KUKA KRL program: f1_Kuka_APT217T02S17.SRC

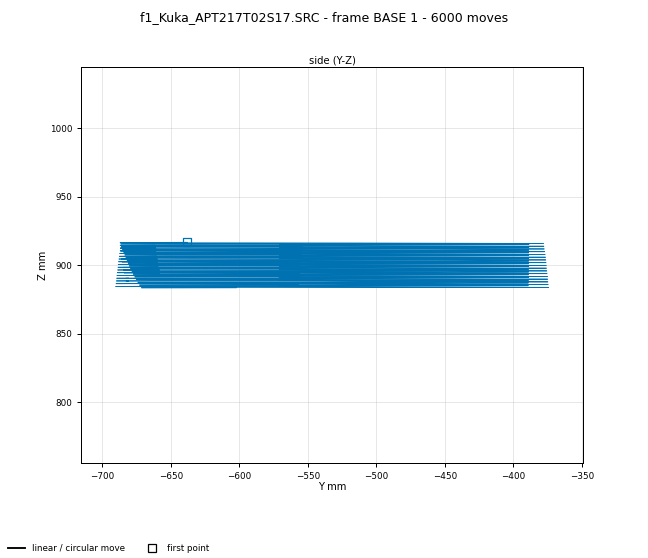
[picture p0: tool path of f1_Kuka_APT217T02S17.SRC in frame BASE 1, 6000 of 6001 moves have a stored position in this frame; points joined in program order, loops and branches not executed]
&ACCESS RVP
&REL 2
&PARAM TEMPLATE = C:\KRC\Roboter\Template\vorgabe
&PARAM EDITMASK = *
DEF f1_Kuka_APT217T02S17()


;FOLD INI;%{PE}%V3.2.0,%MKUKATPBASIS,%CINIT,%VCOMMON,%P
  ;FOLD BAS INI;%{E}%V3.2.0,%MKUKATPBASIS,%CINIT,%VINIT,%P
    GLOBAL INTERRUPT DECL 3 WHEN $STOPMESS==TRUE DO IR_STOPM ( )
    INTERRUPT ON 3
    BAS (#INITMOV,0 )
  ;ENDFOLD (BAS INI)
  ;FOLD USER INI;%{E}%V3.2.0,%MKUKATPUSER,%CINIT,%VINIT,%P
    ;Make your modifications here
  ;ENDFOLD (USER INI)
;ENDFOLD (INI)


;*** Make Null PTP Move
  PTP $pos_act

;*** Auto Load The Correct TOOL Data
  $tool=tool_data[2]

;*** Auto Load The Correct BASE Data
  $base=base_data[1]

  $ADVANCE = 5

;*** Restate Last Velocity
MMPM(30000.0)
SetRPM(8000)
LIN {X -0.126,Y -637.858,Z 916.652,A 0.000,B 0.000,C 90.000,E1 333.384} C_DIS
LIN {X 0.038,Y -640.175,Z 916.648,A 0.000,B 0.000,C 90.000,E1 332.615} C_DIS
LIN {X -0.210,Y -643.727,Z 916.641,A 0.000,B 0.000,C 90.000,E1 331.385} C_DIS
LIN {X 0.321,Y -645.721,Z 916.637,A 0.000,B 0.000,C 90.000,E1 330.589} C_DIS
LIN {X -0.408,Y -648.888,Z 916.630,A 0.000,B 0.000,C 90.000,E1 329.410} C_DIS
LIN {X 0.136,Y -651.837,Z 916.623,A 0.000,B 0.000,C 90.000,E1 328.122} C_DIS
LIN {X 0.289,Y -653.811,Z 916.618,A 0.000,B 0.000,C 90.000,E1 327.120} C_DIS
LIN {X -0.089,Y -655.582,Z 916.612,A 0.000,B 0.000,C 90.000,E1 326.167} C_DIS
LIN {X 0.388,Y -657.387,Z 916.605,A 0.000,B 0.000,C 90.000,E1 324.895} C_DIS
LIN {X 0.431,Y -658.697,Z 916.600,A 0.000,B 0.000,C 90.000,E1 323.909} C_DIS
LIN {X -0.041,Y -659.709,Z 916.594,A 0.000,B 0.000,C 90.000,E1 322.970} C_DIS
LIN {X 0.023,Y -660.733,Z 916.589,A 0.000,B 0.000,C 90.000,E1 321.984} C_DIS
LIN {X -0.032,Y -662.440,Z 916.578,A 0.000,B 0.000,C 90.000,E1 320.033} C_DIS
LIN {X -0.057,Y -664.582,Z 916.564,A 0.000,B 0.000,C 90.000,E1 317.595} C_DIS
LIN {X -0.049,Y -665.667,Z 916.559,A 0.000,B 0.000,C 90.000,E1 316.620} C_DIS
LIN {X -0.059,Y -666.244,Z 916.555,A 0.000,B 0.000,C 90.000,E1 315.891} C_DIS
LIN {X -0.039,Y -668.536,Z 916.540,A 0.000,B 0.000,C 90.000,E1 313.218} C_DIS
LIN {X 0.033,Y -669.951,Z 916.532,A 0.000,B 0.000,C 90.000,E1 311.757} C_DIS
LIN {X 0.126,Y -671.036,Z 916.525,A 0.000,B 0.000,C 90.000,E1 310.539} C_DIS
LIN {X 0.333,Y -672.440,Z 916.516,A 0.000,B 0.000,C 90.000,E1 308.830} C_DIS
LIN {X 0.031,Y -673.306,Z 916.509,A 0.000,B 0.000,C 90.000,E1 307.649} C_DIS
LIN {X 0.276,Y -673.966,Z 916.504,A 0.000,B 0.000,C 90.000,E1 306.664} C_DIS
LIN {X -0.286,Y -674.754,Z 916.495,A 0.000,B 0.000,C 90.000,E1 305.025} C_DIS
LIN {X -0.132,Y -675.681,Z 916.484,A 0.000,B 0.000,C 90.000,E1 303.086} C_DIS
LIN {X -0.151,Y -677.053,Z 916.472,A 0.000,B 0.000,C 90.000,E1 300.924} C_DIS
LIN {X 0.092,Y -679.753,Z 916.456,A 0.000,B 0.000,C 90.000,E1 298.025} C_DIS
LIN {X -0.217,Y -682.675,Z 916.444,A 0.000,B 0.000,C 90.000,E1 295.899} C_DIS
LIN {X -0.081,Y -684.395,Z 916.437,A 0.000,B 0.000,C 90.000,E1 294.695} C_DIS
LIN {X -0.413,Y -685.550,Z 916.432,A 0.000,B 0.000,C 90.000,E1 293.770} C_DIS
LIN {X -0.037,Y -686.075,Z 916.428,A 0.000,B 0.000,C 90.000,E1 293.025} C_DIS
LIN {X 0.393,Y -685.871,Z 916.425,A 0.000,B 0.000,C 90.000,E1 292.514} C_DIS
LIN {X -0.289,Y -685.638,Z 916.424,A 0.000,B 0.000,C 90.000,E1 292.333} C_DIS
LIN {X -0.123,Y -683.879,Z 916.421,A 0.000,B 0.000,C 90.000,E1 291.844} C_DIS
LIN {X 0.084,Y -682.792,Z 916.420,A 0.000,B 0.000,C 90.000,E1 291.589} C_DIS
LIN {X 0.184,Y -681.840,Z 916.419,A 0.000,B 0.000,C 90.000,E1 291.461} C_DIS
LIN {X 0.036,Y -680.423,Z 916.419,A 0.000,B 0.000,C 90.000,E1 291.354} C_DIS
LIN {X -0.276,Y -674.342,Z 916.416,A 0.000,B 0.000,C 90.000,E1 290.972} C_DIS
LIN {X -0.222,Y -664.750,Z 916.414,A 0.000,B 0.000,C 90.000,E1 290.482} C_DIS
LIN {X 0.163,Y -661.931,Z 916.413,A 0.000,B 0.000,C 90.000,E1 290.301} C_DIS
LIN {X 0.103,Y -661.883,Z 916.413,A 0.000,B 0.000,C 90.000,E1 290.301} C_DIS
LIN {X -0.077,Y -661.363,Z 916.412,A 0.000,B 0.000,C 90.000,E1 290.248} C_DIS
LIN {X -0.121,Y -661.335,Z 916.412,A 0.000,B 0.000,C 90.000,E1 290.248} C_DIS
LIN {X -0.189,Y -661.291,Z 916.411,A 0.000,B 0.000,C 90.000,E1 290.066} C_DIS
LIN {X -0.073,Y -661.806,Z 916.410,A 0.000,B 0.000,C 90.000,E1 289.812} C_DIS
LIN {X -0.182,Y -662.452,Z 916.409,A 0.000,B 0.000,C 90.000,E1 289.577} C_DIS
LIN {X -0.112,Y -665.086,Z 916.405,A 0.000,B 0.000,C 90.000,E1 288.960} C_DIS
LIN {X -0.111,Y -669.502,Z 916.401,A 0.000,B 0.000,C 90.000,E1 288.109} C_DIS
LIN {X -0.265,Y -671.949,Z 916.398,A 0.000,B 0.000,C 90.000,E1 287.638} C_DIS
LIN {X -0.202,Y -674.243,Z 916.395,A 0.000,B 0.000,C 90.000,E1 287.149} C_DIS
LIN {X 0.270,Y -677.258,Z 916.391,A 0.000,B 0.000,C 90.000,E1 286.386} C_DIS
LIN {X 0.318,Y -679.580,Z 916.387,A 0.000,B 0.000,C 90.000,E1 285.662} C_DIS
LIN {X 0.202,Y -681.424,Z 916.383,A 0.000,B 0.000,C 90.000,E1 284.954} C_DIS
LIN {X 0.107,Y -682.977,Z 916.379,A 0.000,B 0.000,C 90.000,E1 284.245} C_DIS
LIN {X 0.004,Y -684.701,Z 916.374,A 0.000,B 0.000,C 90.000,E1 283.300} C_DIS
LIN {X -0.084,Y -686.073,Z 916.369,A 0.000,B 0.000,C 90.000,E1 282.355} C_DIS
LIN {X -0.284,Y -686.702,Z 916.365,A 0.000,B 0.000,C 90.000,E1 281.658} C_DIS
LIN {X -0.320,Y -686.990,Z 916.362,A 0.000,B 0.000,C 90.000,E1 281.186} C_DIS
LIN {X 0.316,Y -686.962,Z 916.359,A 0.000,B 0.000,C 90.000,E1 280.658} C_DIS
LIN {X 0.151,Y -686.618,Z 916.357,A 0.000,B 0.000,C 90.000,E1 280.197} C_DIS
LIN {X 0.129,Y -686.308,Z 916.355,A 0.000,B 0.000,C 90.000,E1 279.962} C_DIS
LIN {X -0.035,Y -685.373,Z 916.353,A 0.000,B 0.000,C 90.000,E1 279.500} C_DIS
LIN {X -0.092,Y -683.965,Z 916.350,A 0.000,B 0.000,C 90.000,E1 279.029} C_DIS
LIN {X -0.267,Y -682.163,Z 916.348,A 0.000,B 0.000,C 90.000,E1 278.568} C_DIS
LIN {X 0.174,Y -678.948,Z 916.344,A 0.000,B 0.000,C 90.000,E1 277.814} C_DIS
LIN {X -0.170,Y -674.663,Z 916.339,A 0.000,B 0.000,C 90.000,E1 277.004} C_DIS
LIN {X 0.105,Y -670.562,Z 916.335,A 0.000,B 0.000,C 90.000,E1 276.258} C_DIS
LIN {X -0.152,Y -667.548,Z 916.332,A 0.000,B 0.000,C 90.000,E1 275.796} C_DIS
LIN {X 0.147,Y -663.221,Z 916.329,A 0.000,B 0.000,C 90.000,E1 275.163} C_DIS
LIN {X -0.158,Y -659.457,Z 916.326,A 0.000,B 0.000,C 90.000,E1 274.702} C_DIS
LIN {X 0.118,Y -655.403,Z 916.323,A 0.000,B 0.000,C 90.000,E1 274.188} C_DIS
LIN {X -0.237,Y -650.891,Z 916.321,A 0.000,B 0.000,C 90.000,E1 273.726} C_DIS
LIN {X 0.033,Y -644.710,Z 916.317,A 0.000,B 0.000,C 90.000,E1 273.094} C_DIS
LIN {X 0.003,Y -638.004,Z 916.314,A 0.000,B 0.000,C 90.000,E1 272.522} C_DIS
LIN {X 0.237,Y -630.908,Z 916.311,A 0.000,B 0.000,C 90.000,E1 271.949} C_DIS
LIN {X -0.302,Y -623.315,Z 916.308,A 0.000,B 0.000,C 90.000,E1 271.489} C_DIS
LIN {X -0.112,Y -617.098,Z 916.306,A 0.000,B 0.000,C 90.000,E1 271.088} C_DIS
LIN {X -0.233,Y -610.802,Z 916.304,A 0.000,B 0.000,C 90.000,E1 270.745} C_DIS
LIN {X -0.206,Y -603.986,Z 916.302,A 0.000,B 0.000,C 90.000,E1 270.401} C_DIS
LIN {X 0.120,Y -597.215,Z 916.300,A 0.000,B 0.000,C 90.000,E1 270.057} C_DIS
LIN {X 0.222,Y -591.868,Z 916.299,A 0.000,B 0.000,C 90.000,E1 269.828} C_DIS
LIN {X -0.037,Y -586.277,Z 916.298,A 0.000,B 0.000,C 90.000,E1 269.656} C_DIS
LIN {X 0.001,Y -578.952,Z 916.297,A 0.000,B 0.000,C 90.000,E1 269.427} C_DIS
LIN {X -0.131,Y -571.158,Z 916.296,A 0.000,B 0.000,C 90.000,E1 269.255} C_DIS
LIN {X -0.099,Y -564.308,Z 916.295,A 0.000,B 0.000,C 90.000,E1 269.141} C_DIS
LIN {X -0.044,Y -552.233,Z 916.295,A 0.000,B 0.000,C 90.000,E1 269.026} C_DIS
LIN {X 0.198,Y -548.996,Z 916.294,A 0.000,B 0.000,C 90.000,E1 268.912} C_DIS
LIN {X -0.230,Y -548.179,Z 916.294,A 0.000,B 0.000,C 90.000,E1 268.912} C_DIS
LIN {X -0.086,Y -545.297,Z 916.293,A 0.000,B 0.000,C 90.000,E1 268.682} C_DIS
LIN {X -0.118,Y -545.280,Z 916.293,A 0.000,B 0.000,C 90.000,E1 268.682} C_DIS
LIN {X 0.231,Y -544.006,Z 916.291,A 0.000,B 0.000,C 90.000,E1 268.282} C_DIS
LIN {X -0.084,Y -542.250,Z 916.282,A 0.000,B 0.000,C 90.000,E1 266.788} C_DIS
LIN {X 0.262,Y -540.038,Z 916.266,A 0.000,B 0.000,C 90.000,E1 263.913} C_DIS
LIN {X -0.077,Y -538.982,Z 916.258,A 0.000,B 0.000,C 90.000,E1 262.527} C_DIS
LIN {X 0.094,Y -537.773,Z 916.251,A 0.000,B 0.000,C 90.000,E1 261.084} C_DIS
LIN {X -0.214,Y -536.376,Z 916.243,A 0.000,B 0.000,C 90.000,E1 259.690} C_DIS
LIN {X 0.020,Y -535.047,Z 916.236,A 0.000,B 0.000,C 90.000,E1 258.522} C_DIS
LIN {X -0.191,Y -532.946,Z 916.227,A 0.000,B 0.000,C 90.000,E1 256.825} C_DIS
LIN {X 0.144,Y -531.230,Z 916.219,A 0.000,B 0.000,C 90.000,E1 255.353} C_DIS
LIN {X -0.221,Y -528.389,Z 916.206,A 0.000,B 0.000,C 90.000,E1 253.087} C_DIS
LIN {X 0.146,Y -526.961,Z 916.200,A 0.000,B 0.000,C 90.000,E1 251.891} C_DIS
LIN {X -0.014,Y -524.300,Z 916.188,A 0.000,B 0.000,C 90.000,E1 249.880} C_DIS
LIN {X 0.123,Y -522.391,Z 916.180,A 0.000,B 0.000,C 90.000,E1 248.411} C_DIS
LIN {X 0.264,Y -520.853,Z 916.174,A 0.000,B 0.000,C 90.000,E1 247.230} C_DIS
LIN {X 0.051,Y -518.689,Z 916.166,A 0.000,B 0.000,C 90.000,E1 245.793} C_DIS
LIN {X 0.145,Y -515.996,Z 916.156,A 0.000,B 0.000,C 90.000,E1 244.024} C_DIS
LIN {X -0.062,Y -514.213,Z 916.149,A 0.000,B 0.000,C 90.000,E1 242.871} C_DIS
LIN {X -0.060,Y -511.194,Z 916.139,A 0.000,B 0.000,C 90.000,E1 241.101} C_DIS
LIN {X 0.208,Y -507.461,Z 916.128,A 0.000,B 0.000,C 90.000,E1 238.997} C_DIS
LIN {X 0.052,Y -505.866,Z 916.123,A 0.000,B 0.000,C 90.000,E1 238.122} C_DIS
LIN {X -0.121,Y -504.124,Z 916.118,A 0.000,B 0.000,C 90.000,E1 237.248} C_DIS
LIN {X 0.262,Y -501.504,Z 916.111,A 0.000,B 0.000,C 90.000,E1 236.008} C_DIS
LIN {X 0.068,Y -498.202,Z 916.103,A 0.000,B 0.000,C 90.000,E1 234.529} C_DIS
LIN {X 0.086,Y -492.885,Z 916.090,A 0.000,B 0.000,C 90.000,E1 232.110} C_DIS
LIN {X 0.021,Y -489.445,Z 916.081,A 0.000,B 0.000,C 90.000,E1 230.598} C_DIS
LIN {X -0.038,Y -485.311,Z 916.071,A 0.000,B 0.000,C 90.000,E1 228.771} C_DIS
LIN {X -0.061,Y -480.572,Z 916.059,A 0.000,B 0.000,C 90.000,E1 226.620} C_DIS
LIN {X -0.243,Y -477.858,Z 916.052,A 0.000,B 0.000,C 90.000,E1 225.405} C_DIS
LIN {X -0.014,Y -474.320,Z 916.044,A 0.000,B 0.000,C 90.000,E1 223.824} C_DIS
LIN {X 0.005,Y -469.406,Z 916.031,A 0.000,B 0.000,C 90.000,E1 221.634} C_DIS
LIN {X -0.021,Y -463.936,Z 916.017,A 0.000,B 0.000,C 90.000,E1 219.116} C_DIS
LIN {X 0.037,Y -460.623,Z 916.009,A 0.000,B 0.000,C 90.000,E1 217.523} C_DIS
LIN {X 0.133,Y -456.514,Z 915.998,A 0.000,B 0.000,C 90.000,E1 215.598} C_DIS
LIN {X 0.147,Y -453.128,Z 915.989,A 0.000,B 0.000,C 90.000,E1 213.992} C_DIS
LIN {X -0.157,Y -449.462,Z 915.980,A 0.000,B 0.000,C 90.000,E1 212.418} C_DIS
LIN {X -0.150,Y -445.960,Z 915.971,A 0.000,B 0.000,C 90.000,E1 210.797} C_DIS
LIN {X -0.003,Y -441.643,Z 915.960,A 0.000,B 0.000,C 90.000,E1 208.821} C_DIS
LIN {X -0.035,Y -438.778,Z 915.953,A 0.000,B 0.000,C 90.000,E1 207.513} C_DIS
LIN {X -0.077,Y -434.437,Z 915.942,A 0.000,B 0.000,C 90.000,E1 205.540} C_DIS
LIN {X -0.030,Y -431.536,Z 915.935,A 0.000,B 0.000,C 90.000,E1 204.207} C_DIS
LIN {X 0.166,Y -426.424,Z 915.922,A 0.000,B 0.000,C 90.000,E1 201.844} C_DIS
LIN {X 0.087,Y -422.781,Z 915.912,A 0.000,B 0.000,C 90.000,E1 200.174} C_DIS
LIN {X 0.148,Y -417.354,Z 915.897,A 0.000,B 0.000,C 90.000,E1 197.457} C_DIS
LIN {X -0.115,Y -414.058,Z 915.888,A 0.000,B 0.000,C 90.000,E1 195.788} C_DIS
LIN {X -0.045,Y -410.566,Z 915.878,A 0.000,B 0.000,C 90.000,E1 194.064} C_DIS
LIN {X -0.121,Y -405.687,Z 915.865,A 0.000,B 0.000,C 90.000,E1 191.658} C_DIS
LIN {X -0.011,Y -402.292,Z 915.855,A 0.000,B 0.000,C 90.000,E1 189.905} C_DIS
LIN {X -0.083,Y -397.378,Z 915.841,A 0.000,B 0.000,C 90.000,E1 187.466} C_DIS
LIN {X 0.029,Y -393.315,Z 915.830,A 0.000,B 0.000,C 90.000,E1 185.334} C_DIS
LIN {X -0.085,Y -388.932,Z 915.816,A 0.000,B 0.000,C 90.000,E1 182.865} C_DIS
LIN {X -0.151,Y -385.959,Z 915.806,A 0.000,B 0.000,C 90.000,E1 181.088} C_DIS
LIN {X -0.081,Y -380.437,Z 915.786,A 0.000,B 0.000,C 90.000,E1 177.478} C_DIS
LIN {X -0.056,Y -379.094,Z 915.780,A 0.000,B 0.000,C 90.000,E1 176.388} C_DIS
LIN {X 0.084,Y -378.445,Z 915.776,A 0.000,B 0.000,C 90.000,E1 175.641} C_DIS
LIN {X -0.051,Y -378.213,Z 915.774,A 0.000,B 0.000,C 90.000,E1 175.298} C_DIS
LIN {X 0.044,Y -378.084,Z 915.769,A 0.000,B 0.000,C 90.000,E1 174.375} C_DIS
LIN {X -0.026,Y -378.161,Z 915.768,A 0.000,B 0.000,C 90.000,E1 174.204} C_DIS
LIN {X 0.097,Y -378.414,Z 915.767,A 0.000,B 0.000,C 90.000,E1 173.970} C_DIS
LIN {X -0.077,Y -378.824,Z 915.764,A 0.000,B 0.000,C 90.000,E1 173.451} C_DIS
LIN {X 0.128,Y -379.882,Z 915.761,A 0.000,B 0.000,C 90.000,E1 172.875} C_DIS
LIN {X 0.056,Y -380.113,Z 915.760,A 0.000,B 0.000,C 90.000,E1 172.704} C_DIS
LIN {X -0.023,Y -381.256,Z 915.758,A 0.000,B 0.000,C 90.000,E1 172.356} C_DIS
LIN {X -0.095,Y -381.987,Z 915.757,A 0.000,B 0.000,C 90.000,E1 172.186} C_DIS
LIN {X -0.089,Y -385.404,Z 915.753,A 0.000,B 0.000,C 90.000,E1 171.602} C_DIS
LIN {X -0.159,Y -386.668,Z 915.752,A 0.000,B 0.000,C 90.000,E1 171.432} C_DIS
LIN {X 0.137,Y -391.555,Z 915.749,A 0.000,B 0.000,C 90.000,E1 170.849} C_DIS
LIN {X 0.042,Y -398.395,Z 915.746,A 0.000,B 0.000,C 90.000,E1 170.274} C_DIS
LIN {X 0.183,Y -418.889,Z 915.738,A 0.000,B 0.000,C 90.000,E1 168.870} C_DIS
LIN {X -0.129,Y -426.813,Z 915.735,A 0.000,B 0.000,C 90.000,E1 168.342} C_DIS
LIN {X -0.046,Y -436.131,Z 915.731,A 0.000,B 0.000,C 90.000,E1 167.589} C_DIS
LIN {X 0.118,Y -442.311,Z 915.728,A 0.000,B 0.000,C 90.000,E1 167.061} C_DIS
LIN {X -0.067,Y -455.872,Z 915.722,A 0.000,B 0.000,C 90.000,E1 165.880} C_DIS
LIN {X 0.233,Y -468.313,Z 915.715,A 0.000,B 0.000,C 90.000,E1 164.574} C_DIS
LIN {X -0.018,Y -473.746,Z 915.711,A 0.000,B 0.000,C 90.000,E1 164.031} C_DIS
LIN {X -0.152,Y -484.248,Z 915.705,A 0.000,B 0.000,C 90.000,E1 162.834} C_DIS
LIN {X -0.017,Y -490.256,Z 915.700,A 0.000,B 0.000,C 90.000,E1 162.054} C_DIS
LIN {X -0.074,Y -497.174,Z 915.695,A 0.000,B 0.000,C 90.000,E1 161.148} C_DIS
LIN {X 0.144,Y -502.648,Z 915.691,A 0.000,B 0.000,C 90.000,E1 160.369} C_DIS
LIN {X -0.159,Y -511.136,Z 915.684,A 0.000,B 0.000,C 90.000,E1 159.209} C_DIS
LIN {X -0.112,Y -516.078,Z 915.680,A 0.000,B 0.000,C 90.000,E1 158.465} C_DIS
LIN {X 0.300,Y -522.071,Z 915.675,A 0.000,B 0.000,C 90.000,E1 157.539} C_DIS
LIN {X 0.324,Y -530.498,Z 915.668,A 0.000,B 0.000,C 90.000,E1 156.230} C_DIS
LIN {X -0.124,Y -533.252,Z 915.666,A 0.000,B 0.000,C 90.000,E1 155.845} C_DIS
LIN {X 0.134,Y -537.693,Z 915.662,A 0.000,B 0.000,C 90.000,E1 155.101} C_DIS
LIN {X -0.061,Y -542.155,Z 915.658,A 0.000,B 0.000,C 90.000,E1 154.409} C_DIS
LIN {X -0.101,Y -550.359,Z 915.650,A 0.000,B 0.000,C 90.000,E1 152.999} C_DIS
LIN {X 0.037,Y -552.775,Z 915.648,A 0.000,B 0.000,C 90.000,E1 152.564} C_DIS
LIN {X 0.161,Y -558.858,Z 915.641,A 0.000,B 0.000,C 90.000,E1 151.435} C_DIS
LIN {X 0.009,Y -565.034,Z 915.635,A 0.000,B 0.000,C 90.000,E1 150.205} C_DIS
LIN {X -0.170,Y -570.374,Z 915.628,A 0.000,B 0.000,C 90.000,E1 149.125} C_DIS
LIN {X 0.052,Y -576.717,Z 915.621,A 0.000,B 0.000,C 90.000,E1 147.740} C_DIS
LIN {X 0.187,Y -580.374,Z 915.616,A 0.000,B 0.000,C 90.000,E1 146.914} C_DIS
LIN {X -0.271,Y -585.063,Z 915.610,A 0.000,B 0.000,C 90.000,E1 145.881} C_DIS
LIN {X -0.139,Y -590.655,Z 915.603,A 0.000,B 0.000,C 90.000,E1 144.529} C_DIS
LIN {X 0.359,Y -594.950,Z 915.597,A 0.000,B 0.000,C 90.000,E1 143.417} C_DIS
LIN {X 0.196,Y -600.029,Z 915.590,A 0.000,B 0.000,C 90.000,E1 142.110} C_DIS
LIN {X -0.029,Y -608.431,Z 915.578,A 0.000,B 0.000,C 90.000,E1 140.033} C_DIS
LIN {X -0.159,Y -614.759,Z 915.569,A 0.000,B 0.000,C 90.000,E1 138.485} C_DIS
LIN {X 0.347,Y -620.060,Z 915.562,A 0.000,B 0.000,C 90.000,E1 137.148} C_DIS
LIN {X -0.063,Y -626.543,Z 915.554,A 0.000,B 0.000,C 90.000,E1 135.648} C_DIS
LIN {X 0.206,Y -631.735,Z 915.547,A 0.000,B 0.000,C 90.000,E1 134.352} C_DIS
LIN {X 0.125,Y -636.887,Z 915.540,A 0.000,B 0.000,C 90.000,E1 133.095} C_DIS
LIN {X 0.217,Y -640.998,Z 915.534,A 0.000,B 0.000,C 90.000,E1 132.081} C_DIS
LIN {X -0.142,Y -645.938,Z 915.527,A 0.000,B 0.000,C 90.000,E1 130.862} C_DIS
LIN {X -0.426,Y -650.812,Z 915.520,A 0.000,B 0.000,C 90.000,E1 129.644} C_DIS
LIN {X -0.139,Y -657.437,Z 915.510,A 0.000,B 0.000,C 90.000,E1 127.890} C_DIS
LIN {X -0.143,Y -662.051,Z 915.504,A 0.000,B 0.000,C 90.000,E1 126.664} C_DIS
LIN {X -0.079,Y -666.435,Z 915.497,A 0.000,B 0.000,C 90.000,E1 125.438} C_DIS
LIN {X 0.213,Y -670.660,Z 915.490,A 0.000,B 0.000,C 90.000,E1 124.199} C_DIS
LIN {X 0.057,Y -673.731,Z 915.485,A 0.000,B 0.000,C 90.000,E1 123.245} C_DIS
LIN {X -0.058,Y -676.467,Z 915.479,A 0.000,B 0.000,C 90.000,E1 122.291} C_DIS
LIN {X -0.142,Y -678.905,Z 915.474,A 0.000,B 0.000,C 90.000,E1 121.337} C_DIS
LIN {X -0.205,Y -681.038,Z 915.469,A 0.000,B 0.000,C 90.000,E1 120.384} C_DIS
LIN {X 0.003,Y -682.799,Z 915.463,A 0.000,B 0.000,C 90.000,E1 119.411} C_DIS
LIN {X 0.243,Y -684.380,Z 915.458,A 0.000,B 0.000,C 90.000,E1 118.437} C_DIS
LIN {X 0.287,Y -685.334,Z 915.454,A 0.000,B 0.000,C 90.000,E1 117.719} C_DIS
LIN {X -0.054,Y -686.123,Z 915.449,A 0.000,B 0.000,C 90.000,E1 116.796} C_DIS
LIN {X 0.136,Y -686.609,Z 915.442,A 0.000,B 0.000,C 90.000,E1 115.591} C_DIS
LIN {X 0.113,Y -686.610,Z 915.437,A 0.000,B 0.000,C 90.000,E1 114.643} C_DIS
LIN {X -0.131,Y -686.362,Z 915.433,A 0.000,B 0.000,C 90.000,E1 113.951} C_DIS
LIN {X 0.088,Y -686.187,Z 915.432,A 0.000,B 0.000,C 90.000,E1 113.695} C_DIS
LIN {X 0.251,Y -685.416,Z 915.429,A 0.000,B 0.000,C 90.000,E1 113.206} C_DIS
LIN {X -0.165,Y -684.930,Z 915.428,A 0.000,B 0.000,C 90.000,E1 113.003} C_DIS
LIN {X 0.093,Y -681.933,Z 915.424,A 0.000,B 0.000,C 90.000,E1 112.386} C_DIS
LIN {X -0.064,Y -681.154,Z 915.424,A 0.000,B 0.000,C 90.000,E1 112.280} C_DIS
LIN {X 0.036,Y -679.980,Z 915.423,A 0.000,B 0.000,C 90.000,E1 112.153} C_DIS
LIN {X -0.049,Y -675.165,Z 915.421,A 0.000,B 0.000,C 90.000,E1 111.844} C_DIS
LIN {X 0.343,Y -673.565,Z 915.421,A 0.000,B 0.000,C 90.000,E1 111.716} C_DIS
LIN {X -0.138,Y -671.671,Z 915.420,A 0.000,B 0.000,C 90.000,E1 111.663} C_DIS
LIN {X -0.195,Y -669.497,Z 915.420,A 0.000,B 0.000,C 90.000,E1 111.589} C_DIS
LIN {X 0.075,Y -662.092,Z 915.419,A 0.000,B 0.000,C 90.000,E1 111.408} C_DIS
LIN {X -0.353,Y -659.835,Z 915.419,A 0.000,B 0.000,C 90.000,E1 111.408} C_DIS
LIN {X 0.325,Y -649.462,Z 915.418,A 0.000,B 0.000,C 90.000,E1 111.280} C_DIS
LIN {X -0.137,Y -640.390,Z 915.418,A 0.000,B 0.000,C 90.000,E1 111.280} C_DIS
LIN {X 0.041,Y -633.213,Z 915.418,A 0.000,B 0.000,C 90.000,E1 111.173} C_DIS
LIN {X -0.269,Y -627.334,Z 915.417,A 0.000,B 0.000,C 90.000,E1 111.099} C_DIS
LIN {X 0.265,Y -621.712,Z 915.416,A 0.000,B 0.000,C 90.000,E1 110.918} C_DIS
LIN {X -0.162,Y -614.292,Z 915.415,A 0.000,B 0.000,C 90.000,E1 110.737} C_DIS
LIN {X 0.222,Y -607.266,Z 915.414,A 0.000,B 0.000,C 90.000,E1 110.429} C_DIS
LIN {X 0.126,Y -604.232,Z 915.413,A 0.000,B 0.000,C 90.000,E1 110.301} C_DIS
LIN {X -0.041,Y -597.919,Z 915.411,A 0.000,B 0.000,C 90.000,E1 109.993} C_DIS
LIN {X -0.041,Y -581.000,Z 915.405,A 0.000,B 0.000,C 90.000,E1 108.906} C_DIS
LIN {X 0.321,Y -579.541,Z 915.405,A 0.000,B 0.000,C 90.000,E1 108.779} C_DIS
LIN {X -0.068,Y -572.884,Z 915.403,A 0.000,B 0.000,C 90.000,E1 108.471} C_DIS
LIN {X 0.259,Y -563.917,Z 915.401,A 0.000,B 0.000,C 90.000,E1 108.055} C_DIS
LIN {X 0.007,Y -557.301,Z 915.399,A 0.000,B 0.000,C 90.000,E1 107.819} C_DIS
LIN {X 0.264,Y -555.523,Z 915.398,A 0.000,B 0.000,C 90.000,E1 107.692} C_DIS
LIN {X -0.046,Y -554.039,Z 915.398,A 0.000,B 0.000,C 90.000,E1 107.583} C_DIS
LIN {X -0.085,Y -554.015,Z 915.398,A 0.000,B 0.000,C 90.000,E1 107.583} C_DIS
LIN {X -0.004,Y -553.661,Z 915.396,A 0.000,B 0.000,C 90.000,E1 107.275} C_DIS
LIN {X -0.171,Y -553.838,Z 915.391,A 0.000,B 0.000,C 90.000,E1 106.315} C_DIS
LIN {X -0.087,Y -554.313,Z 915.384,A 0.000,B 0.000,C 90.000,E1 105.190} C_DIS
LIN {X 0.102,Y -555.375,Z 915.372,A 0.000,B 0.000,C 90.000,E1 102.939} C_DIS
LIN {X 0.067,Y -556.899,Z 915.360,A 0.000,B 0.000,C 90.000,E1 100.715} C_DIS
LIN {X 0.238,Y -558.114,Z 915.350,A 0.000,B 0.000,C 90.000,E1 99.029} C_DIS
LIN {X 0.214,Y -559.092,Z 915.343,A 0.000,B 0.000,C 90.000,E1 97.644} C_DIS
LIN {X 0.003,Y -559.681,Z 915.338,A 0.000,B 0.000,C 90.000,E1 96.834} C_DIS
LIN {X 0.170,Y -560.802,Z 915.327,A 0.000,B 0.000,C 90.000,E1 94.878} C_DIS
LIN {X 0.142,Y -561.497,Z 915.320,A 0.000,B 0.000,C 90.000,E1 93.498} C_DIS
LIN {X 0.091,Y -562.172,Z 915.312,A 0.000,B 0.000,C 90.000,E1 92.121} C_DIS
LIN {X 0.151,Y -562.787,Z 915.303,A 0.000,B 0.000,C 90.000,E1 90.458} C_DIS
LIN {X 0.002,Y -563.052,Z 915.297,A 0.000,B 0.000,C 90.000,E1 89.370} C_DIS
LIN {X 0.078,Y -563.406,Z 915.287,A 0.000,B 0.000,C 90.000,E1 87.707} C_DIS
LIN {X -0.045,Y -563.625,Z 915.281,A 0.000,B 0.000,C 90.000,E1 86.617} C_DIS
LIN {X 0.075,Y -563.903,Z 915.272,A 0.000,B 0.000,C 90.000,E1 84.951} C_DIS
LIN {X 0.248,Y -564.169,Z 915.263,A 0.000,B 0.000,C 90.000,E1 83.280} C_DIS
LIN {X -0.062,Y -564.539,Z 915.254,A 0.000,B 0.000,C 90.000,E1 81.659} C_DIS
LIN {X 0.189,Y -565.090,Z 915.245,A 0.000,B 0.000,C 90.000,E1 79.982} C_DIS
LIN {X 0.092,Y -565.820,Z 915.235,A 0.000,B 0.000,C 90.000,E1 78.342} C_DIS
LIN {X 0.189,Y -566.878,Z 915.225,A 0.000,B 0.000,C 90.000,E1 76.408} C_DIS
LIN {X 0.089,Y -567.666,Z 915.217,A 0.000,B 0.000,C 90.000,E1 75.046} C_DIS
LIN {X 0.328,Y -568.516,Z 915.208,A 0.000,B 0.000,C 90.000,E1 73.378} C_DIS
LIN {X 0.033,Y -569.213,Z 915.199,A 0.000,B 0.000,C 90.000,E1 71.764} C_DIS
LIN {X 0.111,Y -569.773,Z 915.190,A 0.000,B 0.000,C 90.000,E1 70.115} C_DIS
LIN {X 0.207,Y -570.193,Z 915.181,A 0.000,B 0.000,C 90.000,E1 68.465} C_DIS
LIN {X -0.007,Y -570.504,Z 915.171,A 0.000,B 0.000,C 90.000,E1 66.847} C_DIS
LIN {X 0.128,Y -570.704,Z 915.161,A 0.000,B 0.000,C 90.000,E1 64.921} C_DIS
LIN {X 0.223,Y -570.771,Z 915.150,A 0.000,B 0.000,C 90.000,E1 62.999} C_DIS
LIN {X 0.151,Y -570.728,Z 915.143,A 0.000,B 0.000,C 90.000,E1 61.641} C_DIS
LIN {X 0.071,Y -570.705,Z 915.135,A 0.000,B 0.000,C 90.000,E1 60.284} C_DIS
LIN {X -0.051,Y -570.523,Z 915.129,A 0.000,B 0.000,C 90.000,E1 59.203} C_DIS
LIN {X -0.289,Y -570.414,Z 915.124,A 0.000,B 0.000,C 90.000,E1 58.408} C_DIS
LIN {X -0.162,Y -569.643,Z 915.115,A 0.000,B 0.000,C 90.000,E1 56.755} C_DIS
LIN {X -0.171,Y -568.940,Z 915.108,A 0.000,B 0.000,C 90.000,E1 55.388} C_DIS
LIN {X -0.123,Y -568.335,Z 915.103,A 0.000,B 0.000,C 90.000,E1 54.562} C_DIS
LIN {X -0.089,Y -567.280,Z 915.097,A 0.000,B 0.000,C 90.000,E1 53.463} C_DIS
LIN {X 0.050,Y -566.019,Z 915.091,A 0.000,B 0.000,C 90.000,E1 52.351} C_DIS
LIN {X 0.059,Y -564.626,Z 915.085,A 0.000,B 0.000,C 90.000,E1 51.251} C_DIS
LIN {X 0.047,Y -562.855,Z 915.079,A 0.000,B 0.000,C 90.000,E1 50.150} C_DIS
LIN {X 0.277,Y -561.369,Z 915.074,A 0.000,B 0.000,C 90.000,E1 49.299} C_DIS
LIN {X 0.037,Y -560.309,Z 915.071,A 0.000,B 0.000,C 90.000,E1 48.771} C_DIS
LIN {X -0.091,Y -557.742,Z 915.065,A 0.000,B 0.000,C 90.000,E1 47.676} C_DIS
LIN {X 0.053,Y -556.318,Z 915.062,A 0.000,B 0.000,C 90.000,E1 47.106} C_DIS
LIN {X -0.191,Y -553.860,Z 915.057,A 0.000,B 0.000,C 90.000,E1 46.296} C_DIS
LIN {X -0.061,Y -551.166,Z 915.052,A 0.000,B 0.000,C 90.000,E1 45.445} C_DIS
LIN {X -0.028,Y -550.233,Z 915.051,A 0.000,B 0.000,C 90.000,E1 45.162} C_DIS
LIN {X -0.327,Y -547.016,Z 915.046,A 0.000,B 0.000,C 90.000,E1 44.352} C_DIS
LIN {X -0.088,Y -544.098,Z 915.042,A 0.000,B 0.000,C 90.000,E1 43.623} C_DIS
LIN {X -0.075,Y -541.595,Z 915.039,A 0.000,B 0.000,C 90.000,E1 43.056} C_DIS
LIN {X -0.263,Y -538.117,Z 915.035,A 0.000,B 0.000,C 90.000,E1 42.366} C_DIS
LIN {X 0.100,Y -535.202,Z 915.032,A 0.000,B 0.000,C 90.000,E1 41.757} C_DIS
LIN {X -0.312,Y -532.038,Z 915.029,A 0.000,B 0.000,C 90.000,E1 41.229} C_DIS
LIN {X 0.164,Y -527.753,Z 915.025,A 0.000,B 0.000,C 90.000,E1 40.458} C_DIS
LIN {X 0.106,Y -524.083,Z 915.022,A 0.000,B 0.000,C 90.000,E1 39.886} C_DIS
LIN {X -0.097,Y -518.344,Z 915.017,A 0.000,B 0.000,C 90.000,E1 39.036} C_DIS
LIN {X -0.090,Y -513.122,Z 915.013,A 0.000,B 0.000,C 90.000,E1 38.302} C_DIS
LIN {X -0.237,Y -508.757,Z 915.010,A 0.000,B 0.000,C 90.000,E1 37.729} C_DIS
LIN {X 0.184,Y -505.350,Z 915.007,A 0.000,B 0.000,C 90.000,E1 37.237} C_DIS
LIN {X -0.025,Y -500.467,Z 915.004,A 0.000,B 0.000,C 90.000,E1 36.664} C_DIS
LIN {X 0.123,Y -496.856,Z 915.001,A 0.000,B 0.000,C 90.000,E1 36.217} C_DIS
LIN {X -0.091,Y -490.347,Z 914.997,A 0.000,B 0.000,C 90.000,E1 35.518} C_DIS
LIN {X -0.203,Y -483.346,Z 914.993,A 0.000,B 0.000,C 90.000,E1 34.818} C_DIS
LIN {X -0.069,Y -477.565,Z 914.990,A 0.000,B 0.000,C 90.000,E1 34.246} C_DIS
LIN {X 0.147,Y -467.323,Z 914.985,A 0.000,B 0.000,C 90.000,E1 33.293} C_DIS
LIN {X 0.192,Y -459.706,Z 914.981,A 0.000,B 0.000,C 90.000,E1 32.625} C_DIS
LIN {X 0.235,Y -447.533,Z 914.976,A 0.000,B 0.000,C 90.000,E1 31.592} C_DIS
LIN {X 0.050,Y -436.600,Z 914.971,A 0.000,B 0.000,C 90.000,E1 30.718} C_DIS
LIN {X 0.059,Y -411.333,Z 914.958,A 0.000,B 0.000,C 90.000,E1 28.487} C_DIS
LIN {X 0.065,Y -403.947,Z 914.954,A 0.000,B 0.000,C 90.000,E1 27.769} C_DIS
LIN {X -0.031,Y -398.103,Z 914.951,A 0.000,B 0.000,C 90.000,E1 27.180} C_DIS
LIN {X 0.052,Y -394.686,Z 914.949,A 0.000,B 0.000,C 90.000,E1 26.744} C_DIS
LIN {X 0.067,Y -391.741,Z 914.946,A 0.000,B 0.000,C 90.000,E1 26.283} C_DIS
LIN {X 0.137,Y -389.672,Z 914.943,A 0.000,B 0.000,C 90.000,E1 25.668} C_DIS
LIN {X -0.100,Y -388.805,Z 914.939,A 0.000,B 0.000,C 90.000,E1 25.079} C_DIS
LIN {X 0.144,Y -388.587,Z 914.935,A 0.000,B 0.000,C 90.000,E1 24.335} C_DIS
LIN {X -0.139,Y -389.455,Z 914.927,A 0.000,B 0.000,C 90.000,E1 22.950} C_DIS
LIN {X -0.173,Y -392.936,Z 914.908,A 0.000,B 0.000,C 90.000,E1 19.396} C_DIS
LIN {X -0.087,Y -396.272,Z 914.892,A 0.000,B 0.000,C 90.000,E1 16.551} C_DIS
LIN {X 0.117,Y -400.358,Z 914.874,A 0.000,B 0.000,C 90.000,E1 13.355} C_DIS
LIN {X -0.183,Y -404.475,Z 914.859,A 0.000,B 0.000,C 90.000,E1 10.602} C_DIS
LIN {X -0.085,Y -409.648,Z 914.841,A 0.000,B 0.000,C 90.000,E1 7.466} C_DIS
LIN {X 0.001,Y -415.369,Z 914.824,A 0.000,B 0.000,C 90.000,E1 4.359} C_DIS
LIN {X 0.172,Y -420.335,Z 914.811,A 0.000,B 0.000,C 90.000,E1 1.949} C_DIS
LIN {X -0.156,Y -426.994,Z 914.795,A 0.000,B 0.000,C 90.000,E1 359.141} C_DIS
LIN {X 0.180,Y -431.388,Z 914.786,A 0.000,B 0.000,C 90.000,E1 357.421} C_DIS
LIN {X -0.138,Y -433.210,Z 914.783,A 0.000,B 0.000,C 90.000,E1 356.963} C_DIS
LIN {X -0.075,Y -433.947,Z 914.782,A 0.000,B 0.000,C 90.000,E1 356.788} C_DIS
LIN {X 0.111,Y -437.101,Z 914.779,A 0.000,B 0.000,C 90.000,E1 356.216} C_DIS
LIN {X -0.203,Y -441.820,Z 914.777,A 0.000,B 0.000,C 90.000,E1 355.812} C_DIS
LIN {X 0.133,Y -442.733,Z 914.776,A 0.000,B 0.000,C 90.000,E1 355.698} C_DIS
LIN {X 0.043,Y -446.815,Z 914.775,A 0.000,B 0.000,C 90.000,E1 355.469} C_DIS
LIN {X 0.014,Y -461.833,Z 914.771,A 0.000,B 0.000,C 90.000,E1 354.780} C_DIS
LIN {X -0.160,Y -478.676,Z 914.766,A 0.000,B 0.000,C 90.000,E1 353.970} C_DIS
LIN {X 0.030,Y -490.195,Z 914.763,A 0.000,B 0.000,C 90.000,E1 353.337} C_DIS
LIN {X 0.108,Y -503.374,Z 914.759,A 0.000,B 0.000,C 90.000,E1 352.591} C_DIS
LIN {X -0.138,Y -509.900,Z 914.757,A 0.000,B 0.000,C 90.000,E1 352.243} C_DIS
LIN {X 0.277,Y -519.398,Z 914.754,A 0.000,B 0.000,C 90.000,E1 351.602} C_DIS
LIN {X -0.205,Y -528.490,Z 914.750,A 0.000,B 0.000,C 90.000,E1 351.027} C_DIS
LIN {X 0.068,Y -535.929,Z 914.747,A 0.000,B 0.000,C 90.000,E1 350.443} C_DIS
LIN {X -0.054,Y -543.007,Z 914.744,A 0.000,B 0.000,C 90.000,E1 349.859} C_DIS
LIN {X 0.086,Y -549.702,Z 914.740,A 0.000,B 0.000,C 90.000,E1 349.218} C_DIS
LIN {X -0.026,Y -554.997,Z 914.737,A 0.000,B 0.000,C 90.000,E1 348.701} C_DIS
LIN {X 0.096,Y -558.836,Z 914.735,A 0.000,B 0.000,C 90.000,E1 348.285} C_DIS
LIN {X 0.187,Y -564.823,Z 914.731,A 0.000,B 0.000,C 90.000,E1 347.589} C_DIS
LIN {X 0.144,Y -571.511,Z 914.727,A 0.000,B 0.000,C 90.000,E1 346.769} C_DIS
LIN {X -0.254,Y -577.653,Z 914.722,A 0.000,B 0.000,C 90.000,E1 345.992} C_DIS
LIN {X -0.170,Y -583.228,Z 914.718,A 0.000,B 0.000,C 90.000,E1 345.172} C_DIS
LIN {X 0.122,Y -588.411,Z 914.713,A 0.000,B 0.000,C 90.000,E1 344.338} C_DIS
LIN {X -0.023,Y -592.424,Z 914.709,A 0.000,B 0.000,C 90.000,E1 343.685} C_DIS
LIN {X -0.263,Y -597.692,Z 914.704,A 0.000,B 0.000,C 90.000,E1 342.779} C_DIS
LIN {X 0.097,Y -605.914,Z 914.695,A 0.000,B 0.000,C 90.000,E1 341.167} C_DIS
LIN {X -0.048,Y -611.653,Z 914.689,A 0.000,B 0.000,C 90.000,E1 340.007} C_DIS
LIN {X -0.109,Y -617.032,Z 914.682,A 0.000,B 0.000,C 90.000,E1 338.847} C_DIS
LIN {X 0.157,Y -620.407,Z 914.678,A 0.000,B 0.000,C 90.000,E1 338.050} C_DIS
LIN {X -0.124,Y -624.708,Z 914.672,A 0.000,B 0.000,C 90.000,E1 337.050} C_DIS
LIN {X -0.346,Y -628.656,Z 914.667,A 0.000,B 0.000,C 90.000,E1 336.049} C_DIS
LIN {X 0.321,Y -632.321,Z 914.661,A 0.000,B 0.000,C 90.000,E1 334.973} C_DIS
LIN {X -0.331,Y -636.659,Z 914.654,A 0.000,B 0.000,C 90.000,E1 333.768} C_DIS
LIN {X -0.180,Y -639.104,Z 914.650,A 0.000,B 0.000,C 90.000,E1 332.999} C_DIS
LIN {X -0.005,Y -641.312,Z 914.646,A 0.000,B 0.000,C 90.000,E1 332.231} C_DIS
LIN {X -0.307,Y -644.146,Z 914.640,A 0.000,B 0.000,C 90.000,E1 331.257} C_DIS
LIN {X -0.181,Y -647.431,Z 914.633,A 0.000,B 0.000,C 90.000,E1 329.999} C_DIS
LIN {X -0.081,Y -649.885,Z 914.628,A 0.000,B 0.000,C 90.000,E1 328.997} C_DIS
LIN {X 0.050,Y -652.253,Z 914.622,A 0.000,B 0.000,C 90.000,E1 327.995} C_DIS
LIN {X 0.116,Y -653.743,Z 914.618,A 0.000,B 0.000,C 90.000,E1 327.248} C_DIS
LIN {X -0.260,Y -655.564,Z 914.613,A 0.000,B 0.000,C 90.000,E1 326.294} C_DIS
LIN {X -0.246,Y -657.070,Z 914.607,A 0.000,B 0.000,C 90.000,E1 325.308} C_DIS
LIN {X -0.207,Y -658.427,Z 914.602,A 0.000,B 0.000,C 90.000,E1 324.322} C_DIS
LIN {X -0.097,Y -659.326,Z 914.598,A 0.000,B 0.000,C 90.000,E1 323.577} C_DIS
LIN {X 0.352,Y -661.057,Z 914.588,A 0.000,B 0.000,C 90.000,E1 321.823} C_DIS
LIN {X -0.088,Y -662.609,Z 914.579,A 0.000,B 0.000,C 90.000,E1 320.150} C_DIS
LIN {X 0.336,Y -664.251,Z 914.568,A 0.000,B 0.000,C 90.000,E1 318.162} C_DIS
LIN {X -0.158,Y -665.848,Z 914.560,A 0.000,B 0.000,C 90.000,E1 316.743} C_DIS
LIN {X 0.318,Y -666.461,Z 914.556,A 0.000,B 0.000,C 90.000,E1 315.972} C_DIS
LIN {X -0.111,Y -668.776,Z 914.541,A 0.000,B 0.000,C 90.000,E1 313.338} C_DIS
LIN {X -0.073,Y -670.177,Z 914.533,A 0.000,B 0.000,C 90.000,E1 311.881} C_DIS
LIN {X 0.016,Y -671.235,Z 914.526,A 0.000,B 0.000,C 90.000,E1 310.663} C_DIS
LIN {X -0.207,Y -672.628,Z 914.517,A 0.000,B 0.000,C 90.000,E1 308.991} C_DIS
LIN {X 0.443,Y -673.517,Z 914.510,A 0.000,B 0.000,C 90.000,E1 307.729} C_DIS
LIN {X 0.153,Y -674.204,Z 914.505,A 0.000,B 0.000,C 90.000,E1 306.790} C_DIS
LIN {X -0.005,Y -674.908,Z 914.496,A 0.000,B 0.000,C 90.000,E1 305.358} C_DIS
LIN {X 0.013,Y -675.599,Z 914.488,A 0.000,B 0.000,C 90.000,E1 303.913} C_DIS
LIN {X -0.005,Y -676.822,Z 914.476,A 0.000,B 0.000,C 90.000,E1 301.750} C_DIS
LIN {X -0.011,Y -679.215,Z 914.460,A 0.000,B 0.000,C 90.000,E1 298.871} C_DIS
LIN {X 0.078,Y -682.521,Z 914.446,A 0.000,B 0.000,C 90.000,E1 296.232} C_DIS
LIN {X -0.188,Y -684.596,Z 914.438,A 0.000,B 0.000,C 90.000,E1 294.823} C_DIS
LIN {X 0.387,Y -685.725,Z 914.433,A 0.000,B 0.000,C 90.000,E1 293.823} C_DIS
LIN {X -0.084,Y -686.143,Z 914.430,A 0.000,B 0.000,C 90.000,E1 293.387} C_DIS
LIN {X 0.079,Y -686.327,Z 914.427,A 0.000,B 0.000,C 90.000,E1 292.898} C_DIS
LIN {X -0.386,Y -686.047,Z 914.425,A 0.000,B 0.000,C 90.000,E1 292.461} C_DIS
LIN {X -0.172,Y -685.510,Z 914.423,A 0.000,B 0.000,C 90.000,E1 292.206} C_DIS
LIN {X -0.217,Y -684.596,Z 914.422,A 0.000,B 0.000,C 90.000,E1 291.972} C_DIS
LIN {X -0.007,Y -683.524,Z 914.421,A 0.000,B 0.000,C 90.000,E1 291.716} C_DIS
LIN {X 0.096,Y -682.876,Z 914.420,A 0.000,B 0.000,C 90.000,E1 291.589} C_DIS
LIN {X 0.197,Y -681.934,Z 914.419,A 0.000,B 0.000,C 90.000,E1 291.461} C_DIS
LIN {X 0.048,Y -680.529,Z 914.419,A 0.000,B 0.000,C 90.000,E1 291.354} C_DIS
LIN {X -0.098,Y -674.324,Z 914.417,A 0.000,B 0.000,C 90.000,E1 290.972} C_DIS
LIN {X -0.074,Y -661.997,Z 914.413,A 0.000,B 0.000,C 90.000,E1 290.355} C_DIS
LIN {X -0.133,Y -661.936,Z 914.413,A 0.000,B 0.000,C 90.000,E1 290.355} C_DIS
LIN {X -0.061,Y -661.178,Z 914.413,A 0.000,B 0.000,C 90.000,E1 290.248} C_DIS
LIN {X -0.104,Y -661.174,Z 914.412,A 0.000,B 0.000,C 90.000,E1 290.248} C_DIS
LIN {X 0.102,Y -661.165,Z 914.411,A 0.000,B 0.000,C 90.000,E1 289.993} C_DIS
LIN {X 0.106,Y -662.558,Z 914.408,A 0.000,B 0.000,C 90.000,E1 289.504} C_DIS
LIN {X 0.016,Y -665.920,Z 914.404,A 0.000,B 0.000,C 90.000,E1 288.779} C_DIS
LIN {X -0.181,Y -670.318,Z 914.400,A 0.000,B 0.000,C 90.000,E1 287.946} C_DIS
LIN {X -0.122,Y -672.691,Z 914.397,A 0.000,B 0.000,C 90.000,E1 287.457} C_DIS
LIN {X -0.254,Y -674.935,Z 914.394,A 0.000,B 0.000,C 90.000,E1 286.985} C_DIS
LIN {X -0.174,Y -676.917,Z 914.392,A 0.000,B 0.000,C 90.000,E1 286.496} C_DIS
LIN {X -0.320,Y -679.336,Z 914.388,A 0.000,B 0.000,C 90.000,E1 285.788} C_DIS
LIN {X -0.259,Y -681.198,Z 914.384,A 0.000,B 0.000,C 90.000,E1 285.064} C_DIS
LIN {X 0.300,Y -682.766,Z 914.380,A 0.000,B 0.000,C 90.000,E1 284.300} C_DIS
LIN {X 0.190,Y -684.519,Z 914.374,A 0.000,B 0.000,C 90.000,E1 283.355} C_DIS
LIN {X 0.121,Y -685.567,Z 914.370,A 0.000,B 0.000,C 90.000,E1 282.647} C_DIS
LIN {X -0.067,Y -686.139,Z 914.368,A 0.000,B 0.000,C 90.000,E1 282.187} C_DIS
LIN {X -0.122,Y -686.734,Z 914.364,A 0.000,B 0.000,C 90.000,E1 281.478} C_DIS
LIN {X -0.142,Y -686.888,Z 914.362,A 0.000,B 0.000,C 90.000,E1 281.243} C_DIS
LIN {X -0.311,Y -686.853,Z 914.360,A 0.000,B 0.000,C 90.000,E1 280.782} C_DIS
LIN {X 0.325,Y -686.567,Z 914.357,A 0.000,B 0.000,C 90.000,E1 280.254} C_DIS
LIN {X 0.303,Y -686.322,Z 914.356,A 0.000,B 0.000,C 90.000,E1 280.018} C_DIS
LIN {X 0.138,Y -685.417,Z 914.353,A 0.000,B 0.000,C 90.000,E1 279.557} C_DIS
LIN {X -0.028,Y -684.045,Z 914.351,A 0.000,B 0.000,C 90.000,E1 279.095} C_DIS
LIN {X -0.096,Y -682.340,Z 914.348,A 0.000,B 0.000,C 90.000,E1 278.624} C_DIS
LIN {X -0.237,Y -681.406,Z 914.347,A 0.000,B 0.000,C 90.000,E1 278.398} C_DIS
LIN {X 0.345,Y -679.252,Z 914.344,A 0.000,B 0.000,C 90.000,E1 277.871} C_DIS
LIN {X -0.005,Y -675.626,Z 914.340,A 0.000,B 0.000,C 90.000,E1 277.182} C_DIS
LIN {X -0.308,Y -672.334,Z 914.337,A 0.000,B 0.000,C 90.000,E1 276.606} C_DIS
LIN {X 0.117,Y -669.462,Z 914.334,A 0.000,B 0.000,C 90.000,E1 276.087} C_DIS
LIN {X -0.060,Y -667.150,Z 914.332,A 0.000,B 0.000,C 90.000,E1 275.739} C_DIS
LIN {X 0.322,Y -663.724,Z 914.329,A 0.000,B 0.000,C 90.000,E1 275.220} C_DIS
LIN {X -0.075,Y -658.987,Z 914.326,A 0.000,B 0.000,C 90.000,E1 274.645} C_DIS
LIN {X 0.230,Y -654.892,Z 914.323,A 0.000,B 0.000,C 90.000,E1 274.131} C_DIS
LIN {X -0.128,Y -650.320,Z 914.320,A 0.000,B 0.000,C 90.000,E1 273.669} C_DIS
LIN {X 0.218,Y -645.416,Z 914.318,A 0.000,B 0.000,C 90.000,E1 273.154} C_DIS
LIN {X 0.160,Y -638.709,Z 914.314,A 0.000,B 0.000,C 90.000,E1 272.579} C_DIS
LIN {X -0.146,Y -631.775,Z 914.311,A 0.000,B 0.000,C 90.000,E1 272.064} C_DIS
LIN {X -0.133,Y -624.238,Z 914.309,A 0.000,B 0.000,C 90.000,E1 271.547} C_DIS
LIN {X -0.014,Y -617.953,Z 914.306,A 0.000,B 0.000,C 90.000,E1 271.146} C_DIS
LIN {X -0.253,Y -611.450,Z 914.304,A 0.000,B 0.000,C 90.000,E1 270.802} C_DIS
LIN {X 0.147,Y -602.987,Z 914.302,A 0.000,B 0.000,C 90.000,E1 270.344} C_DIS
LIN {X 0.091,Y -597.942,Z 914.301,A 0.000,B 0.000,C 90.000,E1 270.115} C_DIS
LIN {X 0.014,Y -590.759,Z 914.299,A 0.000,B 0.000,C 90.000,E1 269.828} C_DIS
LIN {X -0.245,Y -583.097,Z 914.298,A 0.000,B 0.000,C 90.000,E1 269.599} C_DIS
LIN {X -0.125,Y -577.613,Z 914.297,A 0.000,B 0.000,C 90.000,E1 269.427} C_DIS
LIN {X 0.258,Y -571.750,Z 914.296,A 0.000,B 0.000,C 90.000,E1 269.255} C_DIS
LIN {X -0.278,Y -565.008,Z 914.295,A 0.000,B 0.000,C 90.000,E1 269.198} C_DIS
LIN {X -0.084,Y -555.104,Z 914.295,A 0.000,B 0.000,C 90.000,E1 269.083} C_DIS
LIN {X 0.271,Y -552.540,Z 914.295,A 0.000,B 0.000,C 90.000,E1 269.026} C_DIS
LIN {X 0.047,Y -549.313,Z 914.294,A 0.000,B 0.000,C 90.000,E1 268.969} C_DIS
LIN {X -0.042,Y -545.247,Z 914.293,A 0.000,B 0.000,C 90.000,E1 268.682} C_DIS
LIN {X -0.074,Y -545.214,Z 914.293,A 0.000,B 0.000,C 90.000,E1 268.682} C_DIS
LIN {X 0.043,Y -544.194,Z 914.291,A 0.000,B 0.000,C 90.000,E1 268.396} C_DIS
LIN {X -0.134,Y -542.815,Z 914.285,A 0.000,B 0.000,C 90.000,E1 267.364} C_DIS
LIN {X 0.232,Y -540.235,Z 914.268,A 0.000,B 0.000,C 90.000,E1 264.204} C_DIS
LIN {X -0.045,Y -538.992,Z 914.258,A 0.000,B 0.000,C 90.000,E1 262.527} C_DIS
LIN {X 0.126,Y -537.753,Z 914.251,A 0.000,B 0.000,C 90.000,E1 261.084} C_DIS
LIN {X -0.182,Y -536.363,Z 914.243,A 0.000,B 0.000,C 90.000,E1 259.690} C_DIS
LIN {X 0.052,Y -535.069,Z 914.236,A 0.000,B 0.000,C 90.000,E1 258.522} C_DIS
LIN {X -0.160,Y -532.985,Z 914.227,A 0.000,B 0.000,C 90.000,E1 256.825} C_DIS
LIN {X -0.165,Y -530.921,Z 914.217,A 0.000,B 0.000,C 90.000,E1 255.102} C_DIS
LIN {X -0.187,Y -528.419,Z 914.206,A 0.000,B 0.000,C 90.000,E1 253.087} C_DIS
LIN {X 0.180,Y -526.995,Z 914.200,A 0.000,B 0.000,C 90.000,E1 251.891} C_DIS
LIN {X 0.021,Y -524.331,Z 914.188,A 0.000,B 0.000,C 90.000,E1 249.880} C_DIS
LIN {X -0.168,Y -522.058,Z 914.179,A 0.000,B 0.000,C 90.000,E1 248.156} C_DIS
LIN {X -0.027,Y -520.421,Z 914.172,A 0.000,B 0.000,C 90.000,E1 246.975} C_DIS
LIN {X 0.086,Y -518.722,Z 914.166,A 0.000,B 0.000,C 90.000,E1 245.793} C_DIS
LIN {X -0.157,Y -515.633,Z 914.154,A 0.000,B 0.000,C 90.000,E1 243.768} C_DIS
LIN {X 0.088,Y -513.747,Z 914.148,A 0.000,B 0.000,C 90.000,E1 242.564} C_DIS
LIN {X -0.022,Y -511.230,Z 914.139,A 0.000,B 0.000,C 90.000,E1 241.101} C_DIS
LIN {X 0.246,Y -507.503,Z 914.128,A 0.000,B 0.000,C 90.000,E1 238.997} C_DIS
LIN {X 0.091,Y -505.914,Z 914.123,A 0.000,B 0.000,C 90.000,E1 238.122} C_DIS
LIN {X 0.228,Y -503.551,Z 914.116,A 0.000,B 0.000,C 90.000,E1 236.914} C_DIS
LIN {X -0.218,Y -500.309,Z 914.108,A 0.000,B 0.000,C 90.000,E1 235.468} C_DIS
LIN {X -0.180,Y -498.262,Z 914.103,A 0.000,B 0.000,C 90.000,E1 234.562} C_DIS
LIN {X -0.143,Y -494.900,Z 914.095,A 0.000,B 0.000,C 90.000,E1 233.050} C_DIS
LIN {X -0.015,Y -492.290,Z 914.088,A 0.000,B 0.000,C 90.000,E1 231.823} C_DIS
LIN {X 0.217,Y -488.809,Z 914.079,A 0.000,B 0.000,C 90.000,E1 230.275} C_DIS
LIN {X -0.172,Y -484.744,Z 914.069,A 0.000,B 0.000,C 90.000,E1 228.485} C_DIS
LIN {X 0.239,Y -479.320,Z 914.056,A 0.000,B 0.000,C 90.000,E1 225.972} C_DIS
LIN {X 0.150,Y -475.818,Z 914.047,A 0.000,B 0.000,C 90.000,E1 224.433} C_DIS
LIN {X -0.010,Y -472.235,Z 914.038,A 0.000,B 0.000,C 90.000,E1 222.894} C_DIS
LIN {X 0.055,Y -469.437,Z 914.031,A 0.000,B 0.000,C 90.000,E1 221.634} C_DIS
LIN {X 0.030,Y -464.000,Z 914.017,A 0.000,B 0.000,C 90.000,E1 219.116} C_DIS
LIN {X 0.089,Y -460.654,Z 914.009,A 0.000,B 0.000,C 90.000,E1 217.523} C_DIS
LIN {X 0.081,Y -457.245,Z 914.000,A 0.000,B 0.000,C 90.000,E1 215.931} C_DIS
LIN {X 0.199,Y -453.192,Z 913.989,A 0.000,B 0.000,C 90.000,E1 213.992} C_DIS
LIN {X -0.103,Y -449.521,Z 913.980,A 0.000,B 0.000,C 90.000,E1 212.418} C_DIS
LIN {X -0.095,Y -446.025,Z 913.971,A 0.000,B 0.000,C 90.000,E1 210.797} C_DIS
LIN {X 0.052,Y -441.707,Z 913.960,A 0.000,B 0.000,C 90.000,E1 208.821} C_DIS
LIN {X 0.021,Y -438.842,Z 913.953,A 0.000,B 0.000,C 90.000,E1 207.513} C_DIS
LIN {X -0.020,Y -434.500,Z 913.942,A 0.000,B 0.000,C 90.000,E1 205.540} C_DIS
LIN {X 0.028,Y -431.602,Z 913.935,A 0.000,B 0.000,C 90.000,E1 204.207} C_DIS
LIN {X -0.170,Y -426.509,Z 913.922,A 0.000,B 0.000,C 90.000,E1 201.897} C_DIS
LIN {X 0.148,Y -422.872,Z 913.912,A 0.000,B 0.000,C 90.000,E1 200.174} C_DIS
LIN {X 0.048,Y -418.094,Z 913.899,A 0.000,B 0.000,C 90.000,E1 197.819} C_DIS
LIN {X 0.164,Y -415.459,Z 913.892,A 0.000,B 0.000,C 90.000,E1 196.441} C_DIS
LIN {X 0.094,Y -413.438,Z 913.886,A 0.000,B 0.000,C 90.000,E1 195.426} C_DIS
LIN {X 0.046,Y -409.944,Z 913.876,A 0.000,B 0.000,C 90.000,E1 193.716} C_DIS
LIN {X 0.039,Y -405.090,Z 913.863,A 0.000,B 0.000,C 90.000,E1 191.299} C_DIS
LIN {X 0.058,Y -401.673,Z 913.853,A 0.000,B 0.000,C 90.000,E1 189.557} C_DIS
LIN {X -0.011,Y -397.483,Z 913.841,A 0.000,B 0.000,C 90.000,E1 187.466} C_DIS
LIN {X -0.024,Y -392.128,Z 913.826,A 0.000,B 0.000,C 90.000,E1 184.645} C_DIS
LIN {X -0.099,Y -388.412,Z 913.814,A 0.000,B 0.000,C 90.000,E1 182.522} C_DIS
LIN {X -0.073,Y -386.078,Z 913.806,A 0.000,B 0.000,C 90.000,E1 181.088} C_DIS
LIN {X 0.120,Y -381.063,Z 913.788,A 0.000,B 0.000,C 90.000,E1 177.822} C_DIS
LIN {X 0.027,Y -379.120,Z 913.780,A 0.000,B 0.000,C 90.000,E1 176.388} C_DIS
LIN {X 0.168,Y -378.378,Z 913.776,A 0.000,B 0.000,C 90.000,E1 175.641} C_DIS
LIN {X -0.075,Y -377.849,Z 913.772,A 0.000,B 0.000,C 90.000,E1 174.951} C_DIS
LIN {X 0.055,Y -377.701,Z 913.768,A 0.000,B 0.000,C 90.000,E1 174.204} C_DIS
LIN {X -0.197,Y -378.021,Z 913.764,A 0.000,B 0.000,C 90.000,E1 173.514} C_DIS
LIN {X 0.044,Y -378.395,Z 913.763,A 0.000,B 0.000,C 90.000,E1 173.280} C_DIS
LIN {X -0.206,Y -379.451,Z 913.759,A 0.000,B 0.000,C 90.000,E1 172.591} C_DIS
LIN {X 0.114,Y -380.446,Z 913.757,A 0.000,B 0.000,C 90.000,E1 172.186} C_DIS
LIN {X 0.143,Y -381.706,Z 913.755,A 0.000,B 0.000,C 90.000,E1 171.837} C_DIS
LIN {X -0.030,Y -385.985,Z 913.751,A 0.000,B 0.000,C 90.000,E1 171.141} C_DIS
LIN {X 0.115,Y -390.830,Z 913.748,A 0.000,B 0.000,C 90.000,E1 170.566} C_DIS
LIN {X 0.053,Y -397.742,Z 913.744,A 0.000,B 0.000,C 90.000,E1 169.982} C_DIS
LIN {X 0.012,Y -416.133,Z 913.738,A 0.000,B 0.000,C 90.000,E1 168.757} C_DIS
LIN {X 0.210,Y -425.799,Z 913.734,A 0.000,B 0.000,C 90.000,E1 168.049} C_DIS
LIN {X -0.030,Y -435.112,Z 913.730,A 0.000,B 0.000,C 90.000,E1 167.353} C_DIS
LIN {X 0.168,Y -442.765,Z 913.726,A 0.000,B 0.000,C 90.000,E1 166.700} C_DIS
LIN {X -0.105,Y -454.483,Z 913.721,A 0.000,B 0.000,C 90.000,E1 165.700} C_DIS
LIN {X -0.037,Y -461.494,Z 913.717,A 0.000,B 0.000,C 90.000,E1 164.991} C_DIS
LIN {X 0.150,Y -467.129,Z 913.713,A 0.000,B 0.000,C 90.000,E1 164.393} C_DIS
LIN {X -0.001,Y -473.961,Z 913.709,A 0.000,B 0.000,C 90.000,E1 163.685} C_DIS
LIN {X -0.017,Y -481.964,Z 913.704,A 0.000,B 0.000,C 90.000,E1 162.779} C_DIS
LIN {X -0.128,Y -486.972,Z 913.701,A 0.000,B 0.000,C 90.000,E1 162.181} C_DIS
LIN {X 0.113,Y -495.094,Z 913.695,A 0.000,B 0.000,C 90.000,E1 161.094} C_DIS
LIN {X -0.161,Y -500.712,Z 913.691,A 0.000,B 0.000,C 90.000,E1 160.369} C_DIS
LIN {X -0.210,Y -510.342,Z 913.683,A 0.000,B 0.000,C 90.000,E1 159.028} C_DIS
LIN {X 0.008,Y -514.272,Z 913.680,A 0.000,B 0.000,C 90.000,E1 158.411} C_DIS
LIN {X 0.228,Y -521.278,Z 913.674,A 0.000,B 0.000,C 90.000,E1 157.358} C_DIS
LIN {X 0.217,Y -527.029,Z 913.670,A 0.000,B 0.000,C 90.000,E1 156.485} C_DIS
LIN {X -0.217,Y -532.533,Z 913.665,A 0.000,B 0.000,C 90.000,E1 155.665} C_DIS
LIN {X -0.251,Y -538.843,Z 913.659,A 0.000,B 0.000,C 90.000,E1 154.665} C_DIS
LIN {X -0.070,Y -542.267,Z 913.656,A 0.000,B 0.000,C 90.000,E1 154.076} C_DIS
LIN {X 0.269,Y -551.399,Z 913.647,A 0.000,B 0.000,C 90.000,E1 152.487} C_DIS
LIN {X -0.018,Y -555.122,Z 913.643,A 0.000,B 0.000,C 90.000,E1 151.820} C_DIS
LIN {X 0.166,Y -557.472,Z 913.641,A 0.000,B 0.000,C 90.000,E1 151.385} C_DIS
LIN {X 0.268,Y -563.716,Z 913.634,A 0.000,B 0.000,C 90.000,E1 150.127} C_DIS
LIN {X -0.214,Y -569.087,Z 913.628,A 0.000,B 0.000,C 90.000,E1 149.076} C_DIS
LIN {X -0.250,Y -573.613,Z 913.623,A 0.000,B 0.000,C 90.000,E1 148.122} C_DIS
LIN {X -0.073,Y -579.261,Z 913.616,A 0.000,B 0.000,C 90.000,E1 146.882} C_DIS
LIN {X -0.133,Y -584.546,Z 913.609,A 0.000,B 0.000,C 90.000,E1 145.674} C_DIS
LIN {X -0.007,Y -590.206,Z 913.602,A 0.000,B 0.000,C 90.000,E1 144.322} C_DIS
LIN {X 0.267,Y -593.509,Z 913.597,A 0.000,B 0.000,C 90.000,E1 143.497} C_DIS
LIN {X 0.076,Y -598.659,Z 913.590,A 0.000,B 0.000,C 90.000,E1 142.190} C_DIS
LIN {X 0.273,Y -607.086,Z 913.578,A 0.000,B 0.000,C 90.000,E1 140.070} C_DIS
LIN {X 0.054,Y -613.464,Z 913.570,A 0.000,B 0.000,C 90.000,E1 138.528} C_DIS
LIN {X 0.128,Y -618.857,Z 913.563,A 0.000,B 0.000,C 90.000,E1 137.229} C_DIS
LIN {X -0.308,Y -625.315,Z 913.554,A 0.000,B 0.000,C 90.000,E1 135.729} C_DIS
LIN {X 0.059,Y -629.589,Z 913.548,A 0.000,B 0.000,C 90.000,E1 134.676} C_DIS
LIN {X -0.058,Y -634.773,Z 913.541,A 0.000,B 0.000,C 90.000,E1 133.419} C_DIS
LIN {X -0.088,Y -639.945,Z 913.534,A 0.000,B 0.000,C 90.000,E1 132.162} C_DIS
LIN {X -0.041,Y -644.948,Z 913.527,A 0.000,B 0.000,C 90.000,E1 130.906} C_DIS
LIN {X 0.149,Y -649.819,Z 913.520,A 0.000,B 0.000,C 90.000,E1 129.644} C_DIS
LIN {X -0.040,Y -655.482,Z 913.512,A 0.000,B 0.000,C 90.000,E1 128.177} C_DIS
LIN {X -0.075,Y -660.179,Z 913.505,A 0.000,B 0.000,C 90.000,E1 126.950} C_DIS
LIN {X -0.089,Y -662.837,Z 913.501,A 0.000,B 0.000,C 90.000,E1 126.217} C_DIS
LIN {X 0.141,Y -667.154,Z 913.494,A 0.000,B 0.000,C 90.000,E1 124.978} C_DIS
LIN {X 0.317,Y -670.527,Z 913.489,A 0.000,B 0.000,C 90.000,E1 123.992} C_DIS
LIN {X 0.005,Y -672.834,Z 913.485,A 0.000,B 0.000,C 90.000,E1 123.293} C_DIS
LIN {X 0.277,Y -674.953,Z 913.481,A 0.000,B 0.000,C 90.000,E1 122.546} C_DIS
LIN {X 0.171,Y -677.408,Z 913.476,A 0.000,B 0.000,C 90.000,E1 121.592} C_DIS
LIN {X -0.048,Y -678.603,Z 913.473,A 0.000,B 0.000,C 90.000,E1 121.131} C_DIS
LIN {X -0.119,Y -680.622,Z 913.468,A 0.000,B 0.000,C 90.000,E1 120.178} C_DIS
LIN {X 0.082,Y -682.336,Z 913.462,A 0.000,B 0.000,C 90.000,E1 119.205} C_DIS
LIN {X 0.103,Y -683.541,Z 913.458,A 0.000,B 0.000,C 90.000,E1 118.487} C_DIS
LIN {X 0.135,Y -684.518,Z 913.454,A 0.000,B 0.000,C 90.000,E1 117.769} C_DIS
LIN {X 0.081,Y -685.315,Z 913.449,A 0.000,B 0.000,C 90.000,E1 116.821} C_DIS
LIN {X 0.128,Y -685.642,Z 913.445,A 0.000,B 0.000,C 90.000,E1 116.104} C_DIS
LIN {X -0.126,Y -685.937,Z 913.441,A 0.000,B 0.000,C 90.000,E1 115.412} C_DIS
LIN {X 0.066,Y -685.784,Z 913.435,A 0.000,B 0.000,C 90.000,E1 114.207} C_DIS
LIN {X -0.402,Y -685.507,Z 913.432,A 0.000,B 0.000,C 90.000,E1 113.770} C_DIS
LIN {X 0.029,Y -684.757,Z 913.429,A 0.000,B 0.000,C 90.000,E1 113.259} C_DIS
LIN {X -0.027,Y -684.298,Z 913.428,A 0.000,B 0.000,C 90.000,E1 113.025} C_DIS
LIN {X -0.397,Y -681.494,Z 913.425,A 0.000,B 0.000,C 90.000,E1 112.461} C_DIS
LIN {X -0.294,Y -680.757,Z 913.424,A 0.000,B 0.000,C 90.000,E1 112.333} C_DIS
LIN {X -0.196,Y -679.645,Z 913.423,A 0.000,B 0.000,C 90.000,E1 112.206} C_DIS
LIN {X -0.029,Y -676.391,Z 913.422,A 0.000,B 0.000,C 90.000,E1 111.972} C_DIS
LIN {X 0.213,Y -671.943,Z 913.420,A 0.000,B 0.000,C 90.000,E1 111.663} C_DIS
LIN {X -0.008,Y -669.532,Z 913.420,A 0.000,B 0.000,C 90.000,E1 111.589} C_DIS
LIN {X 0.149,Y -666.254,Z 913.419,A 0.000,B 0.000,C 90.000,E1 111.482} C_DIS
LIN {X -0.145,Y -661.500,Z 913.419,A 0.000,B 0.000,C 90.000,E1 111.408} C_DIS
LIN {X 0.041,Y -658.414,Z 913.419,A 0.000,B 0.000,C 90.000,E1 111.354} C_DIS
LIN {X -0.005,Y -648.305,Z 913.418,A 0.000,B 0.000,C 90.000,E1 111.280} C_DIS
LIN {X 0.146,Y -640.639,Z 913.418,A 0.000,B 0.000,C 90.000,E1 111.227} C_DIS
LIN {X -0.053,Y -633.356,Z 913.418,A 0.000,B 0.000,C 90.000,E1 111.153} C_DIS
LIN {X -0.003,Y -627.588,Z 913.417,A 0.000,B 0.000,C 90.000,E1 111.046} C_DIS
LIN {X 0.068,Y -620.234,Z 913.416,A 0.000,B 0.000,C 90.000,E1 110.865} C_DIS
LIN {X -0.224,Y -612.926,Z 913.415,A 0.000,B 0.000,C 90.000,E1 110.663} C_DIS
LIN {X 0.046,Y -605.866,Z 913.413,A 0.000,B 0.000,C 90.000,E1 110.355} C_DIS
LIN {X -0.240,Y -598.211,Z 913.411,A 0.000,B 0.000,C 90.000,E1 109.993} C_DIS
LIN {X -0.257,Y -580.984,Z 913.405,A 0.000,B 0.000,C 90.000,E1 108.906} C_DIS
LIN {X -0.254,Y -577.738,Z 913.404,A 0.000,B 0.000,C 90.000,E1 108.725} C_DIS
LIN {X 0.306,Y -572.805,Z 913.403,A 0.000,B 0.000,C 90.000,E1 108.417} C_DIS
LIN {X 0.157,Y -565.618,Z 913.401,A 0.000,B 0.000,C 90.000,E1 108.127} C_DIS
LIN {X -0.173,Y -557.056,Z 913.399,A 0.000,B 0.000,C 90.000,E1 107.819} C_DIS
LIN {X -0.209,Y -555.920,Z 913.399,A 0.000,B 0.000,C 90.000,E1 107.764} C_DIS
LIN {X -0.148,Y -554.281,Z 913.398,A 0.000,B 0.000,C 90.000,E1 107.583} C_DIS
LIN {X -0.190,Y -554.266,Z 913.398,A 0.000,B 0.000,C 90.000,E1 107.583} C_DIS
LIN {X -0.068,Y -553.877,Z 913.396,A 0.000,B 0.000,C 90.000,E1 107.275} C_DIS
LIN {X -0.116,Y -554.128,Z 913.389,A 0.000,B 0.000,C 90.000,E1 106.024} C_DIS
LIN {X 0.241,Y -554.706,Z 913.381,A 0.000,B 0.000,C 90.000,E1 104.592} C_DIS
LIN {X 0.179,Y -555.726,Z 913.370,A 0.000,B 0.000,C 90.000,E1 102.647} C_DIS
LIN {X 0.053,Y -557.278,Z 913.358,A 0.000,B 0.000,C 90.000,E1 100.433} C_DIS
LIN {X 0.246,Y -558.478,Z 913.349,A 0.000,B 0.000,C 90.000,E1 98.746} C_DIS
LIN {X -0.175,Y -559.674,Z 913.340,A 0.000,B 0.000,C 90.000,E1 97.125} C_DIS
LIN {X -0.086,Y -560.639,Z 913.330,A 0.000,B 0.000,C 90.000,E1 95.454} C_DIS
LIN {X -0.114,Y -561.386,Z 913.323,A 0.000,B 0.000,C 90.000,E1 94.073} C_DIS
LIN {X -0.137,Y -562.050,Z 913.315,A 0.000,B 0.000,C 90.000,E1 92.694} C_DIS
LIN {X -0.184,Y -562.606,Z 913.307,A 0.000,B 0.000,C 90.000,E1 91.318} C_DIS
LIN {X 0.226,Y -562.968,Z 913.301,A 0.000,B 0.000,C 90.000,E1 90.172} C_DIS
LIN {X 0.079,Y -563.221,Z 913.295,A 0.000,B 0.000,C 90.000,E1 89.083} C_DIS
LIN {X 0.054,Y -563.529,Z 913.287,A 0.000,B 0.000,C 90.000,E1 87.707} C_DIS
LIN {X 0.034,Y -563.765,Z 913.280,A 0.000,B 0.000,C 90.000,E1 86.331} C_DIS
LIN {X 0.151,Y -564.059,Z 913.271,A 0.000,B 0.000,C 90.000,E1 84.666} C_DIS
LIN {X 0.230,Y -564.284,Z 913.263,A 0.000,B 0.000,C 90.000,E1 83.280} C_DIS
LIN {X -0.078,Y -564.667,Z 913.254,A 0.000,B 0.000,C 90.000,E1 81.659} C_DIS
LIN {X 0.175,Y -565.215,Z 913.245,A 0.000,B 0.000,C 90.000,E1 79.982} C_DIS
LIN {X 0.081,Y -565.944,Z 913.235,A 0.000,B 0.000,C 90.000,E1 78.342} C_DIS
LIN {X -0.164,Y -566.666,Z 913.228,A 0.000,B 0.000,C 90.000,E1 76.992} C_DIS
LIN {X -0.089,Y -567.617,Z 913.219,A 0.000,B 0.000,C 90.000,E1 75.338} C_DIS
LIN {X -0.005,Y -568.443,Z 913.209,A 0.000,B 0.000,C 90.000,E1 73.685} C_DIS
LIN {X -0.133,Y -569.180,Z 913.200,A 0.000,B 0.000,C 90.000,E1 72.054} C_DIS
LIN {X -0.046,Y -569.646,Z 913.193,A 0.000,B 0.000,C 90.000,E1 70.678} C_DIS
LIN {X -0.108,Y -570.026,Z 913.185,A 0.000,B 0.000,C 90.000,E1 69.316} C_DIS
LIN {X 0.168,Y -570.343,Z 913.177,A 0.000,B 0.000,C 90.000,E1 67.922} C_DIS
LIN {X 0.118,Y -570.557,Z 913.170,A 0.000,B 0.000,C 90.000,E1 66.561} C_DIS
LIN {X -0.042,Y -570.734,Z 913.159,A 0.000,B 0.000,C 90.000,E1 64.665} C_DIS
LIN {X 0.224,Y -570.756,Z 913.150,A 0.000,B 0.000,C 90.000,E1 62.999} C_DIS
LIN {X 0.321,Y -570.774,Z 913.144,A 0.000,B 0.000,C 90.000,E1 61.897} C_DIS
LIN {X 0.071,Y -570.659,Z 913.135,A 0.000,B 0.000,C 90.000,E1 60.284} C_DIS
LIN {X 0.123,Y -570.543,Z 913.130,A 0.000,B 0.000,C 90.000,E1 59.459} C_DIS
LIN {X -0.290,Y -570.328,Z 913.124,A 0.000,B 0.000,C 90.000,E1 58.408} C_DIS
LIN {X -0.289,Y -569.678,Z 913.117,A 0.000,B 0.000,C 90.000,E1 57.041} C_DIS
LIN {X -0.105,Y -569.109,Z 913.111,A 0.000,B 0.000,C 90.000,E1 55.928} C_DIS
LIN {X -0.050,Y -568.598,Z 913.106,A 0.000,B 0.000,C 90.000,E1 55.102} C_DIS
LIN {X -0.129,Y -568.204,Z 913.103,A 0.000,B 0.000,C 90.000,E1 54.562} C_DIS
LIN {X -0.097,Y -567.135,Z 913.097,A 0.000,B 0.000,C 90.000,E1 53.463} C_DIS
LIN {X 0.039,Y -565.855,Z 913.091,A 0.000,B 0.000,C 90.000,E1 52.351} C_DIS
LIN {X 0.047,Y -564.431,Z 913.085,A 0.000,B 0.000,C 90.000,E1 51.251} C_DIS
LIN {X -0.070,Y -563.141,Z 913.080,A 0.000,B 0.000,C 90.000,E1 50.436} C_DIS
LIN {X 0.259,Y -561.119,Z 913.074,A 0.000,B 0.000,C 90.000,E1 49.299} C_DIS
LIN {X 0.018,Y -560.044,Z 913.071,A 0.000,B 0.000,C 90.000,E1 48.771} C_DIS
LIN {X 0.223,Y -558.130,Z 913.066,A 0.000,B 0.000,C 90.000,E1 47.919} C_DIS
LIN {X -0.040,Y -556.769,Z 913.063,A 0.000,B 0.000,C 90.000,E1 47.391} C_DIS
LIN {X 0.126,Y -554.364,Z 913.059,A 0.000,B 0.000,C 90.000,E1 46.539} C_DIS
LIN {X -0.134,Y -551.686,Z 913.054,A 0.000,B 0.000,C 90.000,E1 45.729} C_DIS
LIN {X -0.060,Y -549.792,Z 913.051,A 0.000,B 0.000,C 90.000,E1 45.162} C_DIS
LIN {X 0.018,Y -546.535,Z 913.046,A 0.000,B 0.000,C 90.000,E1 44.312} C_DIS
LIN {X 0.067,Y -542.935,Z 913.042,A 0.000,B 0.000,C 90.000,E1 43.461} C_DIS
LIN {X 0.068,Y -540.325,Z 913.038,A 0.000,B 0.000,C 90.000,E1 42.894} C_DIS
LIN {X 0.083,Y -537.529,Z 913.035,A 0.000,B 0.000,C 90.000,E1 42.324} C_DIS
LIN {X 0.043,Y -534.530,Z 913.032,A 0.000,B 0.000,C 90.000,E1 41.757} C_DIS
LIN {X -0.022,Y -531.304,Z 913.029,A 0.000,B 0.000,C 90.000,E1 41.191} C_DIS
LIN {X 0.097,Y -526.966,Z 913.025,A 0.000,B 0.000,C 90.000,E1 40.458} C_DIS
LIN {X 0.220,Y -524.230,Z 913.022,A 0.000,B 0.000,C 90.000,E1 40.011} C_DIS
LIN {X -0.177,Y -517.457,Z 913.017,A 0.000,B 0.000,C 90.000,E1 39.036} C_DIS
LIN {X -0.057,Y -511.072,Z 913.012,A 0.000,B 0.000,C 90.000,E1 38.141} C_DIS
LIN {X 0.002,Y -505.495,Z 913.008,A 0.000,B 0.000,C 90.000,E1 37.397} C_DIS
LIN {X -0.109,Y -499.310,Z 913.004,A 0.000,B 0.000,C 90.000,E1 36.664} C_DIS
LIN {X -0.141,Y -495.424,Z 913.001,A 0.000,B 0.000,C 90.000,E1 36.217} C_DIS
LIN {X -0.095,Y -490.245,Z 912.998,A 0.000,B 0.000,C 90.000,E1 35.644} C_DIS
LIN {X 0.185,Y -483.249,Z 912.994,A 0.000,B 0.000,C 90.000,E1 34.898} C_DIS
LIN {X 0.037,Y -477.453,Z 912.991,A 0.000,B 0.000,C 90.000,E1 34.358} C_DIS
LIN {X 0.074,Y -467.069,Z 912.986,A 0.000,B 0.000,C 90.000,E1 33.420} C_DIS
LIN {X 0.153,Y -459.489,Z 912.982,A 0.000,B 0.000,C 90.000,E1 32.752} C_DIS
LIN {X -0.084,Y -447.212,Z 912.976,A 0.000,B 0.000,C 90.000,E1 31.750} C_DIS
LIN {X -0.009,Y -436.314,Z 912.971,A 0.000,B 0.000,C 90.000,E1 30.846} C_DIS
LIN {X 0.153,Y -419.894,Z 912.964,A 0.000,B 0.000,C 90.000,E1 29.411} C_DIS
LIN {X 0.200,Y -405.235,Z 912.956,A 0.000,B 0.000,C 90.000,E1 28.025} C_DIS
LIN {X -0.065,Y -397.929,Z 912.952,A 0.000,B 0.000,C 90.000,E1 27.308} C_DIS
LIN {X 0.197,Y -394.754,Z 912.950,A 0.000,B 0.000,C 90.000,E1 26.873} C_DIS
LIN {X -0.017,Y -391.580,Z 912.947,A 0.000,B 0.000,C 90.000,E1 26.411} C_DIS
LIN {X 0.197,Y -389.784,Z 912.944,A 0.000,B 0.000,C 90.000,E1 25.848} C_DIS
LIN {X -0.031,Y -388.753,Z 912.939,A 0.000,B 0.000,C 90.000,E1 25.079} C_DIS
LIN {X 0.026,Y -388.630,Z 912.937,A 0.000,B 0.000,C 90.000,E1 24.719} C_DIS
LIN {X 0.062,Y -389.038,Z 912.931,A 0.000,B 0.000,C 90.000,E1 23.643} C_DIS
LIN {X -0.166,Y -392.681,Z 912.910,A 0.000,B 0.000,C 90.000,E1 19.758} C_DIS
LIN {X -0.088,Y -395.951,Z 912.894,A 0.000,B 0.000,C 90.000,E1 16.913} C_DIS
LIN {X 0.093,Y -398.571,Z 912.882,A 0.000,B 0.000,C 90.000,E1 14.773} C_DIS
LIN {X -0.152,Y -401.482,Z 912.870,A 0.000,B 0.000,C 90.000,E1 12.703} C_DIS
LIN {X -0.108,Y -405.129,Z 912.857,A 0.000,B 0.000,C 90.000,E1 10.254} C_DIS
LIN {X -0.008,Y -409.748,Z 912.841,A 0.000,B 0.000,C 90.000,E1 7.466} C_DIS
LIN {X 0.081,Y -414.776,Z 912.826,A 0.000,B 0.000,C 90.000,E1 4.702} C_DIS
LIN {X -0.163,Y -420.433,Z 912.811,A 0.000,B 0.000,C 90.000,E1 2.007} C_DIS
LIN {X -0.036,Y -428.799,Z 912.791,A 0.000,B 0.000,C 90.000,E1 358.453} C_DIS
LIN {X 0.184,Y -431.460,Z 912.786,A 0.000,B 0.000,C 90.000,E1 357.421} C_DIS
LIN {X -0.073,Y -433.883,Z 912.782,A 0.000,B 0.000,C 90.000,E1 356.788} C_DIS
LIN {X -0.077,Y -436.280,Z 912.780,A 0.000,B 0.000,C 90.000,E1 356.331} C_DIS
LIN {X 0.038,Y -437.286,Z 912.779,A 0.000,B 0.000,C 90.000,E1 356.159} C_DIS
LIN {X 0.077,Y -442.593,Z 912.776,A 0.000,B 0.000,C 90.000,E1 355.641} C_DIS
LIN {X 0.100,Y -448.497,Z 912.774,A 0.000,B 0.000,C 90.000,E1 355.298} C_DIS
LIN {X -0.119,Y -461.754,Z 912.771,A 0.000,B 0.000,C 90.000,E1 354.723} C_DIS
LIN {X 0.100,Y -475.255,Z 912.767,A 0.000,B 0.000,C 90.000,E1 354.033} C_DIS
LIN {X 0.196,Y -488.488,Z 912.763,A 0.000,B 0.000,C 90.000,E1 353.337} C_DIS
LIN {X -0.151,Y -501.551,Z 912.759,A 0.000,B 0.000,C 90.000,E1 352.648} C_DIS
LIN {X 0.172,Y -508.032,Z 912.757,A 0.000,B 0.000,C 90.000,E1 352.243} C_DIS
LIN {X 0.102,Y -517.582,Z 912.754,A 0.000,B 0.000,C 90.000,E1 351.659} C_DIS
LIN {X 0.195,Y -526.813,Z 912.750,A 0.000,B 0.000,C 90.000,E1 351.027} C_DIS
LIN {X -0.020,Y -534.327,Z 912.747,A 0.000,B 0.000,C 90.000,E1 350.500} C_DIS
LIN {X -0.156,Y -541.465,Z 912.744,A 0.000,B 0.000,C 90.000,E1 349.926} C_DIS
LIN {X 0.025,Y -548.243,Z 912.741,A 0.000,B 0.000,C 90.000,E1 349.285} C_DIS
LIN {X 0.050,Y -554.777,Z 912.737,A 0.000,B 0.000,C 90.000,E1 348.634} C_DIS
LIN {X 0.082,Y -558.670,Z 912.735,A 0.000,B 0.000,C 90.000,E1 348.229} C_DIS
LIN {X 0.294,Y -564.641,Z 912.731,A 0.000,B 0.000,C 90.000,E1 347.521} C_DIS
LIN {X 0.006,Y -572.461,Z 912.726,A 0.000,B 0.000,C 90.000,E1 346.589} C_DIS
LIN {X -0.276,Y -577.539,Z 912.722,A 0.000,B 0.000,C 90.000,E1 345.936} C_DIS
LIN {X 0.050,Y -582.216,Z 912.718,A 0.000,B 0.000,C 90.000,E1 345.227} C_DIS
LIN {X -0.146,Y -586.648,Z 912.714,A 0.000,B 0.000,C 90.000,E1 344.574} C_DIS
LIN {X 0.186,Y -591.629,Z 912.710,A 0.000,B 0.000,C 90.000,E1 343.740} C_DIS
LIN {X -0.297,Y -597.672,Z 912.704,A 0.000,B 0.000,C 90.000,E1 342.725} C_DIS
LIN {X 0.004,Y -603.868,Z 912.697,A 0.000,B 0.000,C 90.000,E1 341.511} C_DIS
LIN {X -0.022,Y -607.233,Z 912.694,A 0.000,B 0.000,C 90.000,E1 340.859} C_DIS
LIN {X -0.120,Y -612.312,Z 912.688,A 0.000,B 0.000,C 90.000,E1 339.826} C_DIS
LIN {X 0.067,Y -617.105,Z 912.682,A 0.000,B 0.000,C 90.000,E1 338.773} C_DIS
LIN {X 0.338,Y -620.503,Z 912.678,A 0.000,B 0.000,C 90.000,E1 337.975} C_DIS
LIN {X 0.069,Y -623.798,Z 912.674,A 0.000,B 0.000,C 90.000,E1 337.230} C_DIS
LIN {X -0.161,Y -627.823,Z 912.668,A 0.000,B 0.000,C 90.000,E1 336.230} C_DIS
LIN {X -0.340,Y -631.563,Z 912.662,A 0.000,B 0.000,C 90.000,E1 335.229} C_DIS
LIN {X -0.159,Y -635.997,Z 912.655,A 0.000,B 0.000,C 90.000,E1 333.948} C_DIS
LIN {X 0.046,Y -639.273,Z 912.650,A 0.000,B 0.000,C 90.000,E1 332.922} C_DIS
LIN {X 0.291,Y -642.226,Z 912.644,A 0.000,B 0.000,C 90.000,E1 331.897} C_DIS
LIN {X 0.005,Y -645.038,Z 912.638,A 0.000,B 0.000,C 90.000,E1 330.923} C_DIS
LIN {X 0.150,Y -648.289,Z 912.632,A 0.000,B 0.000,C 90.000,E1 329.665} C_DIS
LIN {X 0.262,Y -650.700,Z 912.626,A 0.000,B 0.000,C 90.000,E1 328.663} C_DIS
LIN {X -0.147,Y -653.029,Z 912.621,A 0.000,B 0.000,C 90.000,E1 327.709} C_DIS
LIN {X -0.436,Y -655.364,Z 912.614,A 0.000,B 0.000,C 90.000,E1 326.501} C_DIS
LIN {X 0.115,Y -656.981,Z 912.608,A 0.000,B 0.000,C 90.000,E1 325.468} C_DIS
LIN {X -0.300,Y -658.684,Z 912.601,A 0.000,B 0.000,C 90.000,E1 324.276} C_DIS
LIN {X 0.147,Y -659.850,Z 912.596,A 0.000,B 0.000,C 90.000,E1 323.256} C_DIS
LIN {X -0.270,Y -661.337,Z 912.588,A 0.000,B 0.000,C 90.000,E1 321.823} C_DIS
LIN {X 0.229,Y -662.935,Z 912.578,A 0.000,B 0.000,C 90.000,E1 320.070} C_DIS
LIN {X 0.200,Y -665.111,Z 912.565,A 0.000,B 0.000,C 90.000,E1 317.634} C_DIS
LIN {X -0.277,Y -666.137,Z 912.559,A 0.000,B 0.000,C 90.000,E1 316.701} C_DIS
LIN {X -0.283,Y -666.754,Z 912.555,A 0.000,B 0.000,C 90.000,E1 315.972} C_DIS
LIN {X -0.259,Y -668.421,Z 912.544,A 0.000,B 0.000,C 90.000,E1 314.028} C_DIS
LIN {X 0.260,Y -669.589,Z 912.538,A 0.000,B 0.000,C 90.000,E1 312.771} C_DIS
LIN {X -0.150,Y -670.716,Z 912.531,A 0.000,B 0.000,C 90.000,E1 311.595} C_DIS
LIN {X -0.054,Y -671.581,Z 912.526,A 0.000,B 0.000,C 90.000,E1 310.620} C_DIS
LIN {X 0.167,Y -672.973,Z 912.516,A 0.000,B 0.000,C 90.000,E1 308.910} C_DIS
LIN {X 0.409,Y -674.061,Z 912.508,A 0.000,B 0.000,C 90.000,E1 307.443} C_DIS
LIN {X 0.125,Y -674.673,Z 912.503,A 0.000,B 0.000,C 90.000,E1 306.503} C_DIS
LIN {X 0.124,Y -675.490,Z 912.494,A 0.000,B 0.000,C 90.000,E1 304.818} C_DIS
LIN {X -0.003,Y -676.069,Z 912.487,A 0.000,B 0.000,C 90.000,E1 303.627} C_DIS
LIN {X -0.191,Y -677.184,Z 912.476,A 0.000,B 0.000,C 90.000,E1 301.720} C_DIS
LIN {X 0.258,Y -679.140,Z 912.463,A 0.000,B 0.000,C 90.000,E1 299.283} C_DIS
LIN {X -0.037,Y -682.604,Z 912.447,A 0.000,B 0.000,C 90.000,E1 296.437} C_DIS
LIN {X -0.077,Y -685.001,Z 912.438,A 0.000,B 0.000,C 90.000,E1 294.771} C_DIS
LIN {X -0.119,Y -686.084,Z 912.432,A 0.000,B 0.000,C 90.000,E1 293.823} C_DIS
LIN {X 0.041,Y -686.462,Z 912.430,A 0.000,B 0.000,C 90.000,E1 293.334} C_DIS
LIN {X -0.423,Y -686.599,Z 912.427,A 0.000,B 0.000,C 90.000,E1 292.898} C_DIS
LIN {X 0.009,Y -686.253,Z 912.424,A 0.000,B 0.000,C 90.000,E1 292.386} C_DIS
LIN {X -0.036,Y -685.610,Z 912.423,A 0.000,B 0.000,C 90.000,E1 292.153} C_DIS
LIN {X 0.176,Y -684.585,Z 912.422,A 0.000,B 0.000,C 90.000,E1 291.897} C_DIS
LIN {X 0.132,Y -683.381,Z 912.420,A 0.000,B 0.000,C 90.000,E1 291.663} C_DIS
LIN {X 0.235,Y -682.660,Z 912.420,A 0.000,B 0.000,C 90.000,E1 291.535} C_DIS
LIN {X 0.336,Y -681.587,Z 912.419,A 0.000,B 0.000,C 90.000,E1 291.408} C_DIS
LIN {X -0.199,Y -679.979,Z 912.418,A 0.000,B 0.000,C 90.000,E1 291.334} C_DIS
LIN {X 0.151,Y -676.328,Z 912.417,A 0.000,B 0.000,C 90.000,E1 291.099} C_DIS
LIN {X 0.153,Y -673.473,Z 912.416,A 0.000,B 0.000,C 90.000,E1 290.918} C_DIS
LIN {X -0.184,Y -665.144,Z 912.414,A 0.000,B 0.000,C 90.000,E1 290.556} C_DIS
LIN {X 0.062,Y -661.702,Z 912.413,A 0.000,B 0.000,C 90.000,E1 290.355} C_DIS
LIN {X 0.003,Y -661.633,Z 912.413,A 0.000,B 0.000,C 90.000,E1 290.355} C_DIS
LIN {X 0.237,Y -660.979,Z 912.413,A 0.000,B 0.000,C 90.000,E1 290.248} C_DIS
LIN {X 0.177,Y -660.944,Z 912.413,A 0.000,B 0.000,C 90.000,E1 290.248} C_DIS
LIN {X -0.061,Y -660.915,Z 912.412,A 0.000,B 0.000,C 90.000,E1 290.120} C_DIS
LIN {X -0.004,Y -661.039,Z 912.411,A 0.000,B 0.000,C 90.000,E1 289.993} C_DIS
LIN {X -0.162,Y -662.096,Z 912.409,A 0.000,B 0.000,C 90.000,E1 289.631} C_DIS
LIN {X -0.119,Y -665.219,Z 912.405,A 0.000,B 0.000,C 90.000,E1 288.906} C_DIS
LIN {X -0.258,Y -670.268,Z 912.400,A 0.000,B 0.000,C 90.000,E1 287.946} C_DIS
LIN {X -0.201,Y -672.645,Z 912.397,A 0.000,B 0.000,C 90.000,E1 287.457} C_DIS
LIN {X -0.136,Y -674.881,Z 912.394,A 0.000,B 0.000,C 90.000,E1 286.968} C_DIS
LIN {X -0.254,Y -676.865,Z 912.392,A 0.000,B 0.000,C 90.000,E1 286.496} C_DIS
LIN {X -0.400,Y -679.268,Z 912.388,A 0.000,B 0.000,C 90.000,E1 285.788} C_DIS
LIN {X 0.316,Y -681.121,Z 912.384,A 0.000,B 0.000,C 90.000,E1 285.009} C_DIS
LIN {X 0.217,Y -682.663,Z 912.380,A 0.000,B 0.000,C 90.000,E1 284.300} C_DIS
LIN {X 0.132,Y -684.038,Z 912.376,A 0.000,B 0.000,C 90.000,E1 283.592} C_DIS
LIN {X 0.059,Y -685.144,Z 912.372,A 0.000,B 0.000,C 90.000,E1 282.883} C_DIS
LIN {X -0.007,Y -686.026,Z 912.368,A 0.000,B 0.000,C 90.000,E1 282.175} C_DIS
LIN {X -0.209,Y -686.613,Z 912.364,A 0.000,B 0.000,C 90.000,E1 281.478} C_DIS
LIN {X -0.229,Y -686.735,Z 912.362,A 0.000,B 0.000,C 90.000,E1 281.243} C_DIS
LIN {X 0.277,Y -686.699,Z 912.360,A 0.000,B 0.000,C 90.000,E1 280.725} C_DIS
LIN {X 0.236,Y -686.392,Z 912.357,A 0.000,B 0.000,C 90.000,E1 280.254} C_DIS
LIN {X 0.214,Y -686.117,Z 912.356,A 0.000,B 0.000,C 90.000,E1 280.018} C_DIS
LIN {X 0.047,Y -685.213,Z 912.353,A 0.000,B 0.000,C 90.000,E1 279.557} C_DIS
LIN {X -0.120,Y -683.886,Z 912.351,A 0.000,B 0.000,C 90.000,E1 279.095} C_DIS
LIN {X -0.189,Y -682.197,Z 912.348,A 0.000,B 0.000,C 90.000,E1 278.624} C_DIS
LIN {X -0.329,Y -681.272,Z 912.347,A 0.000,B 0.000,C 90.000,E1 278.398} C_DIS
LIN {X 0.252,Y -679.114,Z 912.344,A 0.000,B 0.000,C 90.000,E1 277.871} C_DIS
LIN {X -0.026,Y -676.151,Z 912.341,A 0.000,B 0.000,C 90.000,E1 277.296} C_DIS
LIN {X -0.323,Y -672.911,Z 912.337,A 0.000,B 0.000,C 90.000,E1 276.720} C_DIS
LIN {X 0.104,Y -670.092,Z 912.335,A 0.000,B 0.000,C 90.000,E1 276.201} C_DIS
LIN {X -0.072,Y -667.866,Z 912.333,A 0.000,B 0.000,C 90.000,E1 275.853} C_DIS
LIN {X 0.227,Y -663.595,Z 912.329,A 0.000,B 0.000,C 90.000,E1 275.220} C_DIS
LIN {X -0.076,Y -659.873,Z 912.326,A 0.000,B 0.000,C 90.000,E1 274.759} C_DIS
LIN {X 0.103,Y -654.690,Z 912.323,A 0.000,B 0.000,C 90.000,E1 274.131} C_DIS
LIN {X -0.256,Y -650.065,Z 912.320,A 0.000,B 0.000,C 90.000,E1 273.669} C_DIS
LIN {X 0.087,Y -645.130,Z 912.318,A 0.000,B 0.000,C 90.000,E1 273.154} C_DIS
LIN {X 0.054,Y -638.415,Z 912.314,A 0.000,B 0.000,C 90.000,E1 272.579} C_DIS
LIN {X 0.305,Y -631.334,Z 912.311,A 0.000,B 0.000,C 90.000,E1 272.007} C_DIS
LIN {X -0.258,Y -623.770,Z 912.309,A 0.000,B 0.000,C 90.000,E1 271.547} C_DIS
LIN {X -0.102,Y -617.527,Z 912.306,A 0.000,B 0.000,C 90.000,E1 271.146} C_DIS
LIN {X -0.134,Y -611.229,Z 912.304,A 0.000,B 0.000,C 90.000,E1 270.802} C_DIS
LIN {X 0.266,Y -602.692,Z 912.302,A 0.000,B 0.000,C 90.000,E1 270.344} C_DIS
LIN {X 0.213,Y -597.636,Z 912.301,A 0.000,B 0.000,C 90.000,E1 270.115} C_DIS
LIN {X 0.149,Y -590.260,Z 912.299,A 0.000,B 0.000,C 90.000,E1 269.828} C_DIS
LIN {X -0.010,Y -584.798,Z 912.298,A 0.000,B 0.000,C 90.000,E1 269.656} C_DIS
LIN {X 0.103,Y -577.343,Z 912.297,A 0.000,B 0.000,C 90.000,E1 269.427} C_DIS
LIN {X -0.083,Y -571.425,Z 912.296,A 0.000,B 0.000,C 90.000,E1 269.312} C_DIS
LIN {X -0.039,Y -564.513,Z 912.296,A 0.000,B 0.000,C 90.000,E1 269.198} C_DIS
LIN {X 0.010,Y -552.423,Z 912.295,A 0.000,B 0.000,C 90.000,E1 269.083} C_DIS
LIN {X -0.207,Y -549.436,Z 912.294,A 0.000,B 0.000,C 90.000,E1 269.026} C_DIS
LIN {X -0.238,Y -549.328,Z 912.294,A 0.000,B 0.000,C 90.000,E1 269.026} C_DIS
LIN {X -0.139,Y -547.412,Z 912.294,A 0.000,B 0.000,C 90.000,E1 268.854} C_DIS
LIN {X -0.010,Y -545.291,Z 912.293,A 0.000,B 0.000,C 90.000,E1 268.682} C_DIS
LIN {X -0.044,Y -545.244,Z 912.293,A 0.000,B 0.000,C 90.000,E1 268.682} C_DIS
LIN {X 0.114,Y -544.095,Z 912.291,A 0.000,B 0.000,C 90.000,E1 268.339} C_DIS
LIN {X 0.080,Y -542.012,Z 912.281,A 0.000,B 0.000,C 90.000,E1 266.502} C_DIS
LIN {X -0.135,Y -540.058,Z 912.266,A 0.000,B 0.000,C 90.000,E1 263.970} C_DIS
LIN {X -0.006,Y -539.028,Z 912.259,A 0.000,B 0.000,C 90.000,E1 262.534} C_DIS
LIN {X 0.234,Y -537.765,Z 912.251,A 0.000,B 0.000,C 90.000,E1 261.084} C_DIS
LIN {X -0.074,Y -536.375,Z 912.243,A 0.000,B 0.000,C 90.000,E1 259.690} C_DIS
LIN {X 0.160,Y -535.116,Z 912.236,A 0.000,B 0.000,C 90.000,E1 258.522} C_DIS
LIN {X -0.051,Y -533.051,Z 912.227,A 0.000,B 0.000,C 90.000,E1 256.825} C_DIS
LIN {X -0.055,Y -530.966,Z 912.217,A 0.000,B 0.000,C 90.000,E1 255.102} C_DIS
LIN {X -0.077,Y -528.463,Z 912.206,A 0.000,B 0.000,C 90.000,E1 253.087} C_DIS
LIN {X -0.210,Y -527.040,Z 912.200,A 0.000,B 0.000,C 90.000,E1 251.945} C_DIS
LIN {X -0.034,Y -524.749,Z 912.190,A 0.000,B 0.000,C 90.000,E1 250.188} C_DIS
LIN {X 0.110,Y -522.873,Z 912.182,A 0.000,B 0.000,C 90.000,E1 248.720} C_DIS
LIN {X -0.069,Y -520.880,Z 912.174,A 0.000,B 0.000,C 90.000,E1 247.283} C_DIS
LIN {X 0.054,Y -519.246,Z 912.167,A 0.000,B 0.000,C 90.000,E1 246.102} C_DIS
LIN {X -0.044,Y -515.719,Z 912.154,A 0.000,B 0.000,C 90.000,E1 243.768} C_DIS
LIN {X 0.094,Y -513.320,Z 912.146,A 0.000,B 0.000,C 90.000,E1 242.281} C_DIS
LIN {X -0.154,Y -511.292,Z 912.140,A 0.000,B 0.000,C 90.000,E1 241.129} C_DIS
LIN {X -0.335,Y -507.563,Z 912.128,A 0.000,B 0.000,C 90.000,E1 239.076} C_DIS
LIN {X 0.206,Y -505.978,Z 912.123,A 0.000,B 0.000,C 90.000,E1 238.122} C_DIS
LIN {X -0.078,Y -503.633,Z 912.116,A 0.000,B 0.000,C 90.000,E1 236.962} C_DIS
LIN {X -0.102,Y -500.456,Z 912.108,A 0.000,B 0.000,C 90.000,E1 235.468} C_DIS
LIN {X 0.244,Y -496.374,Z 912.098,A 0.000,B 0.000,C 90.000,E1 233.623} C_DIS
LIN {X 0.104,Y -492.369,Z 912.088,A 0.000,B 0.000,C 90.000,E1 231.823} C_DIS
LIN {X 0.025,Y -488.888,Z 912.080,A 0.000,B 0.000,C 90.000,E1 230.312} C_DIS
LIN {X -0.050,Y -484.877,Z 912.069,A 0.000,B 0.000,C 90.000,E1 228.485} C_DIS
LIN {X -0.317,Y -479.400,Z 912.056,A 0.000,B 0.000,C 90.000,E1 226.053} C_DIS
LIN {X 0.273,Y -475.903,Z 912.047,A 0.000,B 0.000,C 90.000,E1 224.433} C_DIS
LIN {X -0.207,Y -472.320,Z 912.038,A 0.000,B 0.000,C 90.000,E1 222.933} C_DIS
LIN {X 0.026,Y -468.112,Z 912.028,A 0.000,B 0.000,C 90.000,E1 221.024} C_DIS
LIN {X 0.155,Y -464.084,Z 912.017,A 0.000,B 0.000,C 90.000,E1 219.116} C_DIS
LIN {X 0.215,Y -460.704,Z 912.009,A 0.000,B 0.000,C 90.000,E1 217.523} C_DIS
LIN {X -0.170,Y -458.011,Z 912.002,A 0.000,B 0.000,C 90.000,E1 216.297} C_DIS
LIN {X 0.230,Y -453.944,Z 911.991,A 0.000,B 0.000,C 90.000,E1 214.326} C_DIS
LIN {X 0.139,Y -451.811,Z 911.986,A 0.000,B 0.000,C 90.000,E1 213.372} C_DIS
LIN {X 0.032,Y -446.108,Z 911.971,A 0.000,B 0.000,C 90.000,E1 210.797} C_DIS
LIN {X 0.182,Y -441.790,Z 911.960,A 0.000,B 0.000,C 90.000,E1 208.821} C_DIS
LIN {X -0.015,Y -438.179,Z 911.951,A 0.000,B 0.000,C 90.000,E1 207.206} C_DIS
LIN {X 0.110,Y -434.585,Z 911.942,A 0.000,B 0.000,C 90.000,E1 205.540} C_DIS
LIN {X 0.158,Y -431.690,Z 911.935,A 0.000,B 0.000,C 90.000,E1 204.207} C_DIS
LIN {X -0.038,Y -426.618,Z 911.922,A 0.000,B 0.000,C 90.000,E1 201.897} C_DIS
LIN {X -0.076,Y -422.302,Z 911.910,A 0.000,B 0.000,C 90.000,E1 199.885} C_DIS
LIN {X -0.014,Y -416.932,Z 911.895,A 0.000,B 0.000,C 90.000,E1 197.166} C_DIS
LIN {X -0.168,Y -413.527,Z 911.886,A 0.000,B 0.000,C 90.000,E1 195.481} C_DIS
LIN {X -0.094,Y -409.349,Z 911.875,A 0.000,B 0.000,C 90.000,E1 193.411} C_DIS
LIN {X 0.178,Y -405.227,Z 911.863,A 0.000,B 0.000,C 90.000,E1 191.299} C_DIS
LIN {X -0.198,Y -401.796,Z 911.853,A 0.000,B 0.000,C 90.000,E1 189.613} C_DIS
LIN {X 0.079,Y -397.604,Z 911.842,A 0.000,B 0.000,C 90.000,E1 187.473} C_DIS
LIN {X 0.119,Y -392.261,Z 911.826,A 0.000,B 0.000,C 90.000,E1 184.645} C_DIS
LIN {X -0.043,Y -387.993,Z 911.812,A 0.000,B 0.000,C 90.000,E1 182.178} C_DIS
LIN {X 0.158,Y -384.480,Z 911.800,A 0.000,B 0.000,C 90.000,E1 180.000} C_DIS
LIN {X 0.153,Y -380.684,Z 911.786,A 0.000,B 0.000,C 90.000,E1 177.478} C_DIS
LIN {X 0.179,Y -379.195,Z 911.780,A 0.000,B 0.000,C 90.000,E1 176.388} C_DIS
LIN {X 0.078,Y -377.732,Z 911.772,A 0.000,B 0.000,C 90.000,E1 174.951} C_DIS
LIN {X -0.170,Y -377.487,Z 911.768,A 0.000,B 0.000,C 90.000,E1 174.261} C_DIS
LIN {X -0.047,Y -377.644,Z 911.764,A 0.000,B 0.000,C 90.000,E1 173.514} C_DIS
LIN {X -0.077,Y -377.605,Z 911.763,A 0.000,B 0.000,C 90.000,E1 173.337} C_DIS
LIN {X -0.148,Y -378.523,Z 911.759,A 0.000,B 0.000,C 90.000,E1 172.591} C_DIS
LIN {X 0.174,Y -379.788,Z 911.756,A 0.000,B 0.000,C 90.000,E1 172.008} C_DIS
LIN {X 0.135,Y -381.220,Z 911.754,A 0.000,B 0.000,C 90.000,E1 171.602} C_DIS
LIN {X 0.062,Y -381.960,Z 911.753,A 0.000,B 0.000,C 90.000,E1 171.432} C_DIS
LIN {X -0.039,Y -385.226,Z 911.750,A 0.000,B 0.000,C 90.000,E1 170.905} C_DIS
LIN {X -0.115,Y -388.014,Z 911.747,A 0.000,B 0.000,C 90.000,E1 170.557} C_DIS
LIN {X -0.021,Y -390.417,Z 911.746,A 0.000,B 0.000,C 90.000,E1 170.274} C_DIS
LIN {X 0.037,Y -396.414,Z 911.743,A 0.000,B 0.000,C 90.000,E1 169.746} C_DIS
LIN {X -0.110,Y -414.978,Z 911.736,A 0.000,B 0.000,C 90.000,E1 168.522} C_DIS
LIN {X 0.011,Y -420.026,Z 911.734,A 0.000,B 0.000,C 90.000,E1 168.173} C_DIS
LIN {X 0.163,Y -429.319,Z 911.731,A 0.000,B 0.000,C 90.000,E1 167.465} C_DIS
LIN {X -0.076,Y -437.133,Z 911.727,A 0.000,B 0.000,C 90.000,E1 166.881} C_DIS
LIN {X 0.102,Y -443.312,Z 911.724,A 0.000,B 0.000,C 90.000,E1 166.353} C_DIS
LIN {X 0.190,Y -447.743,Z 911.722,A 0.000,B 0.000,C 90.000,E1 165.936} C_DIS
LIN {X -0.008,Y -450.933,Z 911.721,A 0.000,B 0.000,C 90.000,E1 165.700} C_DIS
LIN {X -0.126,Y -457.996,Z 911.717,A 0.000,B 0.000,C 90.000,E1 165.046} C_DIS
LIN {X 0.122,Y -463.665,Z 911.714,A 0.000,B 0.000,C 90.000,E1 164.448} C_DIS
LIN {X -0.040,Y -473.308,Z 911.708,A 0.000,B 0.000,C 90.000,E1 163.449} C_DIS
LIN {X -0.240,Y -480.013,Z 911.704,A 0.000,B 0.000,C 90.000,E1 162.725} C_DIS
LIN {X -0.140,Y -486.309,Z 911.700,A 0.000,B 0.000,C 90.000,E1 161.945} C_DIS
LIN {X -0.248,Y -493.494,Z 911.695,A 0.000,B 0.000,C 90.000,E1 161.040} C_DIS
LIN {X -0.166,Y -498.149,Z 911.691,A 0.000,B 0.000,C 90.000,E1 160.423} C_DIS
LIN {X -0.159,Y -509.947,Z 911.682,A 0.000,B 0.000,C 90.000,E1 158.773} C_DIS
LIN {X 0.137,Y -518.930,Z 911.675,A 0.000,B 0.000,C 90.000,E1 157.411} C_DIS
LIN {X 0.265,Y -526.705,Z 911.668,A 0.000,B 0.000,C 90.000,E1 156.230} C_DIS
LIN {X 0.074,Y -536.770,Z 911.659,A 0.000,B 0.000,C 90.000,E1 154.665} C_DIS
LIN {X -0.159,Y -542.783,Z 911.654,A 0.000,B 0.000,C 90.000,E1 153.691} C_DIS
LIN {X 0.057,Y -549.510,Z 911.648,A 0.000,B 0.000,C 90.000,E1 152.538} C_DIS
LIN {X -0.234,Y -556.379,Z 911.641,A 0.000,B 0.000,C 90.000,E1 151.307} C_DIS
LIN {X -0.327,Y -562.018,Z 911.634,A 0.000,B 0.000,C 90.000,E1 150.205} C_DIS
LIN {X -0.160,Y -568.133,Z 911.627,A 0.000,B 0.000,C 90.000,E1 148.948} C_DIS
LIN {X -0.207,Y -572.742,Z 911.622,A 0.000,B 0.000,C 90.000,E1 147.995} C_DIS
LIN {X -0.045,Y -578.442,Z 911.615,A 0.000,B 0.000,C 90.000,E1 146.755} C_DIS
LIN {X 0.132,Y -584.346,Z 911.608,A 0.000,B 0.000,C 90.000,E1 145.388} C_DIS
LIN {X 0.060,Y -588.947,Z 911.602,A 0.000,B 0.000,C 90.000,E1 144.322} C_DIS
LIN {X -0.155,Y -592.270,Z 911.597,A 0.000,B 0.000,C 90.000,E1 143.543} C_DIS
LIN {X 0.110,Y -597.534,Z 911.590,A 0.000,B 0.000,C 90.000,E1 142.190} C_DIS
LIN {X 0.277,Y -605.978,Z 911.578,A 0.000,B 0.000,C 90.000,E1 140.070} C_DIS
LIN {X 0.220,Y -611.395,Z 911.571,A 0.000,B 0.000,C 90.000,E1 138.771} C_DIS
LIN {X -0.068,Y -618.934,Z 911.561,A 0.000,B 0.000,C 90.000,E1 136.986} C_DIS
LIN {X -0.362,Y -624.354,Z 911.554,A 0.000,B 0.000,C 90.000,E1 135.729} C_DIS
LIN {X 0.119,Y -627.672,Z 911.550,A 0.000,B 0.000,C 90.000,E1 134.919} C_DIS
LIN {X 0.294,Y -633.883,Z 911.541,A 0.000,B 0.000,C 90.000,E1 133.380} C_DIS
LIN {X -0.089,Y -638.112,Z 911.536,A 0.000,B 0.000,C 90.000,E1 132.405} C_DIS
LIN {X -0.069,Y -643.172,Z 911.529,A 0.000,B 0.000,C 90.000,E1 131.148} C_DIS
LIN {X 0.096,Y -648.048,Z 911.522,A 0.000,B 0.000,C 90.000,E1 129.886} C_DIS
LIN {X -0.160,Y -652.811,Z 911.515,A 0.000,B 0.000,C 90.000,E1 128.669} C_DIS
LIN {X 0.221,Y -658.515,Z 911.507,A 0.000,B 0.000,C 90.000,E1 127.156} C_DIS
LIN {X -0.202,Y -661.218,Z 911.503,A 0.000,B 0.000,C 90.000,E1 126.457} C_DIS
LIN {X -0.037,Y -666.376,Z 911.494,A 0.000,B 0.000,C 90.000,E1 124.978} C_DIS
LIN {X -0.292,Y -670.515,Z 911.488,A 0.000,B 0.000,C 90.000,E1 123.785} C_DIS
LIN {X -0.042,Y -672.769,Z 911.484,A 0.000,B 0.000,C 90.000,E1 123.038} C_DIS
LIN {X 0.071,Y -674.201,Z 911.481,A 0.000,B 0.000,C 90.000,E1 122.546} C_DIS
LIN {X 0.130,Y -677.229,Z 911.474,A 0.000,B 0.000,C 90.000,E1 121.337} C_DIS
LIN {X -0.088,Y -678.349,Z 911.472,A 0.000,B 0.000,C 90.000,E1 120.875} C_DIS
LIN {X 0.237,Y -679.851,Z 911.468,A 0.000,B 0.000,C 90.000,E1 120.129} C_DIS
LIN {X -0.161,Y -681.557,Z 911.462,A 0.000,B 0.000,C 90.000,E1 119.205} C_DIS
LIN {X -0.148,Y -682.763,Z 911.458,A 0.000,B 0.000,C 90.000,E1 118.487} C_DIS
LIN {X 0.088,Y -683.975,Z 911.453,A 0.000,B 0.000,C 90.000,E1 117.513} C_DIS
LIN {X 0.029,Y -684.702,Z 911.448,A 0.000,B 0.000,C 90.000,E1 116.565} C_DIS
LIN {X -0.116,Y -685.181,Z 911.441,A 0.000,B 0.000,C 90.000,E1 115.387} C_DIS
LIN {X -0.230,Y -685.020,Z 911.434,A 0.000,B 0.000,C 90.000,E1 114.207} C_DIS
LIN {X 0.199,Y -684.752,Z 911.432,A 0.000,B 0.000,C 90.000,E1 113.695} C_DIS
LIN {X -0.276,Y -683.979,Z 911.429,A 0.000,B 0.000,C 90.000,E1 113.259} C_DIS
LIN {X -0.067,Y -683.470,Z 911.428,A 0.000,B 0.000,C 90.000,E1 113.003} C_DIS
LIN {X 0.180,Y -680.663,Z 911.424,A 0.000,B 0.000,C 90.000,E1 112.386} C_DIS
LIN {X 0.021,Y -679.790,Z 911.424,A 0.000,B 0.000,C 90.000,E1 112.280} C_DIS
LIN {X 0.118,Y -678.472,Z 911.423,A 0.000,B 0.000,C 90.000,E1 112.153} C_DIS
LIN {X -0.027,Y -675.143,Z 911.422,A 0.000,B 0.000,C 90.000,E1 111.950} C_DIS
LIN {X 0.279,Y -672.593,Z 911.421,A 0.000,B 0.000,C 90.000,E1 111.716} C_DIS
LIN {X -0.099,Y -670.400,Z 911.420,A 0.000,B 0.000,C 90.000,E1 111.642} C_DIS
LIN {X 0.141,Y -665.168,Z 911.419,A 0.000,B 0.000,C 90.000,E1 111.461} C_DIS
LIN {X 0.249,Y -660.866,Z 911.419,A 0.000,B 0.000,C 90.000,E1 111.354} C_DIS
LIN {X -0.020,Y -650.403,Z 911.418,A 0.000,B 0.000,C 90.000,E1 111.280} C_DIS
LIN {X -0.354,Y -639.054,Z 911.418,A 0.000,B 0.000,C 90.000,E1 111.227} C_DIS
LIN {X 0.170,Y -633.250,Z 911.417,A 0.000,B 0.000,C 90.000,E1 111.099} C_DIS
LIN {X 0.387,Y -627.339,Z 911.417,A 0.000,B 0.000,C 90.000,E1 110.972} C_DIS
LIN {X -0.182,Y -619.926,Z 911.416,A 0.000,B 0.000,C 90.000,E1 110.844} C_DIS
LIN {X -0.153,Y -612.608,Z 911.414,A 0.000,B 0.000,C 90.000,E1 110.610} C_DIS
LIN {X 0.095,Y -605.575,Z 911.413,A 0.000,B 0.000,C 90.000,E1 110.301} C_DIS
LIN {X 0.098,Y -599.385,Z 911.411,A 0.000,B 0.000,C 90.000,E1 109.993} C_DIS
LIN {X -0.279,Y -581.267,Z 911.405,A 0.000,B 0.000,C 90.000,E1 108.906} C_DIS
LIN {X 0.165,Y -577.798,Z 911.404,A 0.000,B 0.000,C 90.000,E1 108.671} C_DIS
LIN {X 0.107,Y -572.665,Z 911.402,A 0.000,B 0.000,C 90.000,E1 108.417} C_DIS
LIN {X -0.058,Y -565.188,Z 911.401,A 0.000,B 0.000,C 90.000,E1 108.127} C_DIS
LIN {X -0.221,Y -557.103,Z 911.399,A 0.000,B 0.000,C 90.000,E1 107.819} C_DIS
LIN {X -0.173,Y -555.887,Z 911.399,A 0.000,B 0.000,C 90.000,E1 107.747} C_DIS
LIN {X -0.062,Y -554.524,Z 911.398,A 0.000,B 0.000,C 90.000,E1 107.583} C_DIS
LIN {X -0.105,Y -554.508,Z 911.398,A 0.000,B 0.000,C 90.000,E1 107.583} C_DIS
LIN {X -0.184,Y -554.096,Z 911.396,A 0.000,B 0.000,C 90.000,E1 107.330} C_DIS
LIN {X 0.246,Y -554.994,Z 911.380,A 0.000,B 0.000,C 90.000,E1 104.356} C_DIS
LIN {X 0.192,Y -556.060,Z 911.369,A 0.000,B 0.000,C 90.000,E1 102.411} C_DIS
LIN {X 0.073,Y -557.627,Z 911.357,A 0.000,B 0.000,C 90.000,E1 100.197} C_DIS
LIN {X -0.146,Y -559.004,Z 911.346,A 0.000,B 0.000,C 90.000,E1 98.276} C_DIS
LIN {X -0.155,Y -559.977,Z 911.338,A 0.000,B 0.000,C 90.000,E1 96.891} C_DIS
LIN {X 0.017,Y -561.088,Z 911.327,A 0.000,B 0.000,C 90.000,E1 94.935} C_DIS
LIN {X -0.007,Y -561.762,Z 911.320,A 0.000,B 0.000,C 90.000,E1 93.555} C_DIS
LIN {X -0.055,Y -562.391,Z 911.312,A 0.000,B 0.000,C 90.000,E1 92.178} C_DIS
LIN {X -0.094,Y -562.905,Z 911.304,A 0.000,B 0.000,C 90.000,E1 90.802} C_DIS
LIN {X -0.137,Y -563.306,Z 911.297,A 0.000,B 0.000,C 90.000,E1 89.427} C_DIS
LIN {X -0.056,Y -563.641,Z 911.288,A 0.000,B 0.000,C 90.000,E1 87.764} C_DIS
LIN {X -0.072,Y -563.862,Z 911.280,A 0.000,B 0.000,C 90.000,E1 86.388} C_DIS
LIN {X 0.047,Y -564.170,Z 911.271,A 0.000,B 0.000,C 90.000,E1 84.723} C_DIS
LIN {X -0.024,Y -564.359,Z 911.265,A 0.000,B 0.000,C 90.000,E1 83.628} C_DIS
LIN {X -0.255,Y -564.779,Z 911.254,A 0.000,B 0.000,C 90.000,E1 81.724} C_DIS
LIN {X 0.252,Y -565.423,Z 911.243,A 0.000,B 0.000,C 90.000,E1 79.746} C_DIS
LIN {X 0.222,Y -566.335,Z 911.233,A 0.000,B 0.000,C 90.000,E1 77.825} C_DIS
LIN {X 0.275,Y -567.186,Z 911.223,A 0.000,B 0.000,C 90.000,E1 76.172} C_DIS
LIN {X 0.180,Y -567.964,Z 911.216,A 0.000,B 0.000,C 90.000,E1 74.810} C_DIS
LIN {X -0.121,Y -568.757,Z 911.207,A 0.000,B 0.000,C 90.000,E1 73.196} C_DIS
LIN {X 0.128,Y -569.426,Z 911.198,A 0.000,B 0.000,C 90.000,E1 71.529} C_DIS
LIN {X -0.140,Y -569.840,Z 911.190,A 0.000,B 0.000,C 90.000,E1 70.188} C_DIS
LIN {X 0.336,Y -570.157,Z 911.182,A 0.000,B 0.000,C 90.000,E1 68.773} C_DIS
LIN {X -0.058,Y -570.397,Z 911.176,A 0.000,B 0.000,C 90.000,E1 67.720} C_DIS
LIN {X -0.097,Y -570.596,Z 911.169,A 0.000,B 0.000,C 90.000,E1 66.357} C_DIS
LIN {X -0.077,Y -570.740,Z 911.160,A 0.000,B 0.000,C 90.000,E1 64.717} C_DIS
LIN {X -0.063,Y -570.750,Z 911.150,A 0.000,B 0.000,C 90.000,E1 63.076} C_DIS
LIN {X 0.029,Y -570.782,Z 911.144,A 0.000,B 0.000,C 90.000,E1 61.975} C_DIS
LIN {X -0.005,Y -570.574,Z 911.132,A 0.000,B 0.000,C 90.000,E1 59.793} C_DIS
LIN {X 0.189,Y -570.248,Z 911.125,A 0.000,B 0.000,C 90.000,E1 58.408} C_DIS
LIN {X 0.065,Y -569.773,Z 911.119,A 0.000,B 0.000,C 90.000,E1 57.327} C_DIS
LIN {X 0.052,Y -569.059,Z 911.111,A 0.000,B 0.000,C 90.000,E1 55.960} C_DIS
LIN {X -0.119,Y -568.104,Z 911.103,A 0.000,B 0.000,C 90.000,E1 54.609} C_DIS
LIN {X 0.037,Y -567.050,Z 911.097,A 0.000,B 0.000,C 90.000,E1 53.497} C_DIS
LIN {X 0.060,Y -565.755,Z 911.091,A 0.000,B 0.000,C 90.000,E1 52.396} C_DIS
LIN {X 0.072,Y -564.319,Z 911.085,A 0.000,B 0.000,C 90.000,E1 51.295} C_DIS
LIN {X -0.041,Y -563.035,Z 911.081,A 0.000,B 0.000,C 90.000,E1 50.481} C_DIS
LIN {X -0.072,Y -560.971,Z 911.074,A 0.000,B 0.000,C 90.000,E1 49.380} C_DIS
LIN {X -0.314,Y -559.892,Z 911.071,A 0.000,B 0.000,C 90.000,E1 48.852} C_DIS
LIN {X -0.110,Y -557.963,Z 911.067,A 0.000,B 0.000,C 90.000,E1 48.000} C_DIS
LIN {X 0.003,Y -556.564,Z 911.064,A 0.000,B 0.000,C 90.000,E1 47.433} C_DIS
LIN {X -0.207,Y -554.169,Z 911.059,A 0.000,B 0.000,C 90.000,E1 46.620} C_DIS
LIN {X 0.311,Y -551.449,Z 911.054,A 0.000,B 0.000,C 90.000,E1 45.729} C_DIS
LIN {X -0.006,Y -549.538,Z 911.051,A 0.000,B 0.000,C 90.000,E1 45.202} C_DIS
LIN {X 0.072,Y -546.282,Z 911.047,A 0.000,B 0.000,C 90.000,E1 44.352} C_DIS
LIN {X 0.105,Y -543.931,Z 911.043,A 0.000,B 0.000,C 90.000,E1 43.785} C_DIS
LIN {X -0.063,Y -540.666,Z 911.039,A 0.000,B 0.000,C 90.000,E1 43.095} C_DIS
LIN {X -0.077,Y -537.901,Z 911.036,A 0.000,B 0.000,C 90.000,E1 42.528} C_DIS
LIN {X 0.284,Y -534.933,Z 911.033,A 0.000,B 0.000,C 90.000,E1 41.919} C_DIS
LIN {X 0.038,Y -530.875,Z 911.029,A 0.000,B 0.000,C 90.000,E1 41.229} C_DIS
LIN {X -0.056,Y -527.397,Z 911.026,A 0.000,B 0.000,C 90.000,E1 40.663} C_DIS
LIN {X -0.119,Y -523.754,Z 911.023,A 0.000,B 0.000,C 90.000,E1 40.092} C_DIS
LIN {X -0.114,Y -516.932,Z 911.017,A 0.000,B 0.000,C 90.000,E1 39.072} C_DIS
LIN {X 0.202,Y -511.591,Z 911.013,A 0.000,B 0.000,C 90.000,E1 38.302} C_DIS
LIN {X -0.012,Y -508.292,Z 911.011,A 0.000,B 0.000,C 90.000,E1 37.890} C_DIS
LIN {X 0.275,Y -505.101,Z 911.008,A 0.000,B 0.000,C 90.000,E1 37.443} C_DIS
LIN {X -0.141,Y -498.887,Z 911.004,A 0.000,B 0.000,C 90.000,E1 36.744} C_DIS
LIN {X -0.172,Y -494.958,Z 911.002,A 0.000,B 0.000,C 90.000,E1 36.297} C_DIS
LIN {X 0.108,Y -489.518,Z 910.998,A 0.000,B 0.000,C 90.000,E1 35.678} C_DIS
LIN {X 0.140,Y -483.888,Z 910.995,A 0.000,B 0.000,C 90.000,E1 35.105} C_DIS
LIN {X 0.080,Y -479.596,Z 910.993,A 0.000,B 0.000,C 90.000,E1 34.692} C_DIS
LIN {X 0.087,Y -475.165,Z 910.991,A 0.000,B 0.000,C 90.000,E1 34.278} C_DIS
LIN {X -0.054,Y -464.759,Z 910.985,A 0.000,B 0.000,C 90.000,E1 33.372} C_DIS
LIN {X 0.064,Y -457.100,Z 910.982,A 0.000,B 0.000,C 90.000,E1 32.704} C_DIS
LIN {X 0.108,Y -446.346,Z 910.977,A 0.000,B 0.000,C 90.000,E1 31.799} C_DIS
LIN {X -0.036,Y -435.463,Z 910.972,A 0.000,B 0.000,C 90.000,E1 30.924} C_DIS
LIN {X 0.150,Y -426.330,Z 910.968,A 0.000,B 0.000,C 90.000,E1 30.129} C_DIS
LIN {X -0.264,Y -411.278,Z 910.960,A 0.000,B 0.000,C 90.000,E1 28.821} C_DIS
LIN {X -0.125,Y -398.381,Z 910.953,A 0.000,B 0.000,C 90.000,E1 27.513} C_DIS
LIN {X -0.044,Y -394.744,Z 910.950,A 0.000,B 0.000,C 90.000,E1 27.052} C_DIS
LIN {X -0.023,Y -391.120,Z 910.947,A 0.000,B 0.000,C 90.000,E1 26.437} C_DIS
LIN {X 0.008,Y -389.567,Z 910.944,A 0.000,B 0.000,C 90.000,E1 25.899} C_DIS
LIN {X 0.131,Y -388.734,Z 910.940,A 0.000,B 0.000,C 90.000,E1 25.079} C_DIS
LIN {X -0.006,Y -388.876,Z 910.935,A 0.000,B 0.000,C 90.000,E1 24.207} C_DIS
LIN {X 0.028,Y -389.538,Z 910.929,A 0.000,B 0.000,C 90.000,E1 23.131} C_DIS
LIN {X -0.006,Y -392.997,Z 910.909,A 0.000,B 0.000,C 90.000,E1 19.577} C_DIS
LIN {X 0.083,Y -396.297,Z 910.893,A 0.000,B 0.000,C 90.000,E1 16.732} C_DIS
LIN {X -0.144,Y -399.390,Z 910.879,A 0.000,B 0.000,C 90.000,E1 14.300} C_DIS
LIN {X -0.065,Y -402.344,Z 910.868,A 0.000,B 0.000,C 90.000,E1 12.187} C_DIS
LIN {X 0.095,Y -406.617,Z 910.852,A 0.000,B 0.000,C 90.000,E1 9.378} C_DIS
LIN {X 0.133,Y -411.355,Z 910.837,A 0.000,B 0.000,C 90.000,E1 6.606} C_DIS
LIN {X -0.119,Y -417.223,Z 910.820,A 0.000,B 0.000,C 90.000,E1 3.555} C_DIS
LIN {X 0.100,Y -422.375,Z 910.807,A 0.000,B 0.000,C 90.000,E1 1.146} C_DIS
LIN {X 0.187,Y -431.532,Z 910.786,A 0.000,B 0.000,C 90.000,E1 357.421} C_DIS
LIN {X -0.071,Y -433.875,Z 910.782,A 0.000,B 0.000,C 90.000,E1 356.788} C_DIS
LIN {X 0.112,Y -435.909,Z 910.780,A 0.000,B 0.000,C 90.000,E1 356.331} C_DIS
LIN {X -0.112,Y -437.588,Z 910.778,A 0.000,B 0.000,C 90.000,E1 356.102} C_DIS
LIN {X -0.122,Y -439.994,Z 910.777,A 0.000,B 0.000,C 90.000,E1 355.869} C_DIS
LIN {X -0.058,Y -441.980,Z 910.776,A 0.000,B 0.000,C 90.000,E1 355.641} C_DIS
LIN {X 0.220,Y -443.024,Z 910.775,A 0.000,B 0.000,C 90.000,E1 355.527} C_DIS
LIN {X 0.009,Y -447.218,Z 910.774,A 0.000,B 0.000,C 90.000,E1 355.298} C_DIS
LIN {X 0.220,Y -455.124,Z 910.772,A 0.000,B 0.000,C 90.000,E1 354.894} C_DIS
LIN {X 0.025,Y -462.024,Z 910.770,A 0.000,B 0.000,C 90.000,E1 354.609} C_DIS
LIN {X -0.151,Y -475.563,Z 910.766,A 0.000,B 0.000,C 90.000,E1 353.970} C_DIS
LIN {X -0.138,Y -485.612,Z 910.764,A 0.000,B 0.000,C 90.000,E1 353.451} C_DIS
LIN {X -0.233,Y -500.302,Z 910.759,A 0.000,B 0.000,C 90.000,E1 352.648} C_DIS
LIN {X -0.224,Y -508.404,Z 910.756,A 0.000,B 0.000,C 90.000,E1 352.186} C_DIS
LIN {X -0.229,Y -517.705,Z 910.753,A 0.000,B 0.000,C 90.000,E1 351.602} C_DIS
LIN {X -0.173,Y -526.976,Z 910.750,A 0.000,B 0.000,C 90.000,E1 350.971} C_DIS
LIN {X 0.131,Y -534.449,Z 910.747,A 0.000,B 0.000,C 90.000,E1 350.387} C_DIS
LIN {X 0.121,Y -541.525,Z 910.743,A 0.000,B 0.000,C 90.000,E1 349.803} C_DIS
LIN {X -0.250,Y -547.071,Z 910.741,A 0.000,B 0.000,C 90.000,E1 349.342} C_DIS
LIN {X -0.324,Y -553.689,Z 910.737,A 0.000,B 0.000,C 90.000,E1 348.701} C_DIS
LIN {X 0.172,Y -558.804,Z 910.734,A 0.000,B 0.000,C 90.000,E1 348.117} C_DIS
LIN {X 0.269,Y -564.450,Z 910.731,A 0.000,B 0.000,C 90.000,E1 347.465} C_DIS
LIN {X 0.224,Y -571.218,Z 910.726,A 0.000,B 0.000,C 90.000,E1 346.645} C_DIS
LIN {X -0.313,Y -577.408,Z 910.721,A 0.000,B 0.000,C 90.000,E1 345.880} C_DIS
LIN {X 0.010,Y -582.115,Z 910.718,A 0.000,B 0.000,C 90.000,E1 345.172} C_DIS
LIN {X -0.274,Y -587.449,Z 910.713,A 0.000,B 0.000,C 90.000,E1 344.393} C_DIS
LIN {X 0.140,Y -591.579,Z 910.709,A 0.000,B 0.000,C 90.000,E1 343.685} C_DIS
LIN {X -0.109,Y -596.934,Z 910.704,A 0.000,B 0.000,C 90.000,E1 342.779} C_DIS
LIN {X -0.006,Y -603.244,Z 910.698,A 0.000,B 0.000,C 90.000,E1 341.583} C_DIS
LIN {X -0.153,Y -608.566,Z 910.692,A 0.000,B 0.000,C 90.000,E1 340.550} C_DIS
LIN {X 0.007,Y -612.985,Z 910.687,A 0.000,B 0.000,C 90.000,E1 339.625} C_DIS
LIN {X 0.005,Y -617.184,Z 910.682,A 0.000,B 0.000,C 90.000,E1 338.720} C_DIS
LIN {X 0.258,Y -621.749,Z 910.676,A 0.000,B 0.000,C 90.000,E1 337.667} C_DIS
LIN {X -0.001,Y -624.977,Z 910.672,A 0.000,B 0.000,C 90.000,E1 336.922} C_DIS
LIN {X -0.216,Y -628.909,Z 910.666,A 0.000,B 0.000,C 90.000,E1 335.921} C_DIS
LIN {X -0.354,Y -633.509,Z 910.659,A 0.000,B 0.000,C 90.000,E1 334.665} C_DIS
LIN {X -0.191,Y -637.050,Z 910.654,A 0.000,B 0.000,C 90.000,E1 333.640} C_DIS
LIN {X -0.036,Y -639.447,Z 910.649,A 0.000,B 0.000,C 90.000,E1 332.871} C_DIS
LIN {X 0.208,Y -642.442,Z 910.644,A 0.000,B 0.000,C 90.000,E1 331.847} C_DIS
LIN {X 0.232,Y -645.245,Z 910.638,A 0.000,B 0.000,C 90.000,E1 330.845} C_DIS
LIN {X 0.060,Y -648.503,Z 910.631,A 0.000,B 0.000,C 90.000,E1 329.616} C_DIS
LIN {X 0.169,Y -650.934,Z 910.626,A 0.000,B 0.000,C 90.000,E1 328.614} C_DIS
LIN {X -0.244,Y -653.268,Z 910.620,A 0.000,B 0.000,C 90.000,E1 327.661} C_DIS
LIN {X 0.280,Y -655.157,Z 910.615,A 0.000,B 0.000,C 90.000,E1 326.628} C_DIS
LIN {X -0.079,Y -656.898,Z 910.609,A 0.000,B 0.000,C 90.000,E1 325.674} C_DIS
LIN {X 0.423,Y -658.638,Z 910.602,A 0.000,B 0.000,C 90.000,E1 324.402} C_DIS
LIN {X -0.049,Y -659.833,Z 910.597,A 0.000,B 0.000,C 90.000,E1 323.463} C_DIS
LIN {X -0.422,Y -661.138,Z 910.590,A 0.000,B 0.000,C 90.000,E1 322.271} C_DIS
LIN {X 0.062,Y -662.038,Z 910.585,A 0.000,B 0.000,C 90.000,E1 321.251} C_DIS
LIN {X 0.024,Y -663.243,Z 910.578,A 0.000,B 0.000,C 90.000,E1 320.033} C_DIS
LIN {X 0.026,Y -665.468,Z 910.564,A 0.000,B 0.000,C 90.000,E1 317.595} C_DIS
LIN {X 0.044,Y -666.451,Z 910.559,A 0.000,B 0.000,C 90.000,E1 316.620} C_DIS
LIN {X 0.043,Y -667.108,Z 910.555,A 0.000,B 0.000,C 90.000,E1 315.891} C_DIS
LIN {X 0.077,Y -668.789,Z 910.544,A 0.000,B 0.000,C 90.000,E1 313.947} C_DIS
LIN {X -0.343,Y -669.962,Z 910.537,A 0.000,B 0.000,C 90.000,E1 312.771} C_DIS
LIN {X 0.189,Y -670.862,Z 910.532,A 0.000,B 0.000,C 90.000,E1 311.757} C_DIS
LIN {X -0.220,Y -671.713,Z 910.527,A 0.000,B 0.000,C 90.000,E1 310.825} C_DIS
LIN {X -0.004,Y -673.107,Z 910.517,A 0.000,B 0.000,C 90.000,E1 309.116} C_DIS
LIN {X -0.174,Y -674.418,Z 910.508,A 0.000,B 0.000,C 90.000,E1 307.443} C_DIS
LIN {X 0.088,Y -675.012,Z 910.503,A 0.000,B 0.000,C 90.000,E1 306.457} C_DIS
LIN {X 0.108,Y -675.848,Z 910.493,A 0.000,B 0.000,C 90.000,E1 304.771} C_DIS
LIN {X -0.006,Y -676.421,Z 910.487,A 0.000,B 0.000,C 90.000,E1 303.579} C_DIS
LIN {X 0.223,Y -677.419,Z 910.477,A 0.000,B 0.000,C 90.000,E1 301.878} C_DIS
LIN {X -0.067,Y -678.454,Z 910.469,A 0.000,B 0.000,C 90.000,E1 300.463} C_DIS
LIN {X 0.112,Y -680.823,Z 910.456,A 0.000,B 0.000,C 90.000,E1 298.052} C_DIS
LIN {X 0.346,Y -683.007,Z 910.447,A 0.000,B 0.000,C 90.000,E1 296.360} C_DIS
LIN {X 0.092,Y -685.061,Z 910.439,A 0.000,B 0.000,C 90.000,E1 294.951} C_DIS
LIN {X -0.232,Y -686.199,Z 910.433,A 0.000,B 0.000,C 90.000,E1 294.027} C_DIS
LIN {X 0.206,Y -686.660,Z 910.431,A 0.000,B 0.000,C 90.000,E1 293.515} C_DIS
LIN {X -0.259,Y -686.916,Z 910.428,A 0.000,B 0.000,C 90.000,E1 293.078} C_DIS
LIN {X -0.088,Y -686.646,Z 910.425,A 0.000,B 0.000,C 90.000,E1 292.589} C_DIS
LIN {X 0.129,Y -686.440,Z 910.424,A 0.000,B 0.000,C 90.000,E1 292.333} C_DIS
LIN {X 0.086,Y -685.647,Z 910.423,A 0.000,B 0.000,C 90.000,E1 292.099} C_DIS
LIN {X -0.127,Y -683.225,Z 910.420,A 0.000,B 0.000,C 90.000,E1 291.642} C_DIS
LIN {X -0.277,Y -682.395,Z 910.420,A 0.000,B 0.000,C 90.000,E1 291.535} C_DIS
LIN {X -0.174,Y -681.165,Z 910.419,A 0.000,B 0.000,C 90.000,E1 291.408} C_DIS
LIN {X -0.049,Y -679.323,Z 910.418,A 0.000,B 0.000,C 90.000,E1 291.280} C_DIS
LIN {X 0.229,Y -674.235,Z 910.417,A 0.000,B 0.000,C 90.000,E1 290.972} C_DIS
LIN {X 0.037,Y -671.851,Z 910.416,A 0.000,B 0.000,C 90.000,E1 290.865} C_DIS
LIN {X 0.280,Y -666.460,Z 910.415,A 0.000,B 0.000,C 90.000,E1 290.610} C_DIS
LIN {X -0.071,Y -661.345,Z 910.413,A 0.000,B 0.000,C 90.000,E1 290.375} C_DIS
LIN {X 0.100,Y -661.303,Z 910.413,A 0.000,B 0.000,C 90.000,E1 290.355} C_DIS
LIN {X -0.227,Y -660.747,Z 910.413,A 0.000,B 0.000,C 90.000,E1 290.301} C_DIS
LIN {X -0.286,Y -660.727,Z 910.413,A 0.000,B 0.000,C 90.000,E1 290.301} C_DIS
LIN {X 0.271,Y -660.826,Z 910.411,A 0.000,B 0.000,C 90.000,E1 289.993} C_DIS
LIN {X 0.111,Y -661.943,Z 910.409,A 0.000,B 0.000,C 90.000,E1 289.631} C_DIS
LIN {X 0.183,Y -663.914,Z 910.406,A 0.000,B 0.000,C 90.000,E1 289.141} C_DIS
LIN {X -0.014,Y -666.301,Z 910.404,A 0.000,B 0.000,C 90.000,E1 288.671} C_DIS
LIN {X 0.071,Y -671.352,Z 910.398,A 0.000,B 0.000,C 90.000,E1 287.692} C_DIS
LIN {X -0.132,Y -674.732,Z 910.394,A 0.000,B 0.000,C 90.000,E1 286.985} C_DIS
LIN {X -0.055,Y -676.714,Z 910.392,A 0.000,B 0.000,C 90.000,E1 286.496} C_DIS
LIN {X -0.201,Y -679.140,Z 910.388,A 0.000,B 0.000,C 90.000,E1 285.788} C_DIS
LIN {X -0.143,Y -680.990,Z 910.384,A 0.000,B 0.000,C 90.000,E1 285.064} C_DIS
LIN {X -0.278,Y -683.054,Z 910.378,A 0.000,B 0.000,C 90.000,E1 284.120} C_DIS
LIN {X 0.303,Y -684.328,Z 910.374,A 0.000,B 0.000,C 90.000,E1 283.355} C_DIS
LIN {X 0.210,Y -685.641,Z 910.369,A 0.000,B 0.000,C 90.000,E1 282.411} C_DIS
LIN {X 0.004,Y -686.320,Z 910.365,A 0.000,B 0.000,C 90.000,E1 281.715} C_DIS
LIN {X -0.036,Y -686.582,Z 910.362,A 0.000,B 0.000,C 90.000,E1 281.243} C_DIS
LIN {X -0.207,Y -686.546,Z 910.360,A 0.000,B 0.000,C 90.000,E1 280.782} C_DIS
LIN {X -0.248,Y -686.219,Z 910.357,A 0.000,B 0.000,C 90.000,E1 280.310} C_DIS
LIN {X -0.272,Y -685.958,Z 910.356,A 0.000,B 0.000,C 90.000,E1 280.074} C_DIS
LIN {X 0.236,Y -685.053,Z 910.353,A 0.000,B 0.000,C 90.000,E1 279.557} C_DIS
LIN {X 0.067,Y -683.797,Z 910.351,A 0.000,B 0.000,C 90.000,E1 279.095} C_DIS
LIN {X -0.003,Y -682.157,Z 910.348,A 0.000,B 0.000,C 90.000,E1 278.624} C_DIS
LIN {X -0.143,Y -681.246,Z 910.347,A 0.000,B 0.000,C 90.000,E1 278.398} C_DIS
LIN {X -0.329,Y -679.094,Z 910.344,A 0.000,B 0.000,C 90.000,E1 277.936} C_DIS
LIN {X 0.158,Y -676.168,Z 910.341,A 0.000,B 0.000,C 90.000,E1 277.296} C_DIS
LIN {X -0.140,Y -672.935,Z 910.337,A 0.000,B 0.000,C 90.000,E1 276.720} C_DIS
LIN {X 0.287,Y -670.123,Z 910.335,A 0.000,B 0.000,C 90.000,E1 276.201} C_DIS
LIN {X 0.027,Y -667.071,Z 910.332,A 0.000,B 0.000,C 90.000,E1 275.739} C_DIS
LIN {X 0.319,Y -662.714,Z 910.329,A 0.000,B 0.000,C 90.000,E1 275.106} C_DIS
LIN {X 0.104,Y -659.936,Z 910.327,A 0.000,B 0.000,C 90.000,E1 274.759} C_DIS
LIN {X 0.295,Y -654.747,Z 910.323,A 0.000,B 0.000,C 90.000,E1 274.131} C_DIS
LIN {X -0.051,Y -650.110,Z 910.320,A 0.000,B 0.000,C 90.000,E1 273.669} C_DIS
LIN {X 0.284,Y -645.142,Z 910.318,A 0.000,B 0.000,C 90.000,E1 273.154} C_DIS
LIN {X 0.251,Y -638.445,Z 910.315,A 0.000,B 0.000,C 90.000,E1 272.579} C_DIS
LIN {X -0.071,Y -631.399,Z 910.311,A 0.000,B 0.000,C 90.000,E1 272.064} C_DIS
LIN {X 0.042,Y -623.929,Z 910.309,A 0.000,B 0.000,C 90.000,E1 271.547} C_DIS
LIN {X 0.183,Y -617.668,Z 910.307,A 0.000,B 0.000,C 90.000,E1 271.146} C_DIS
LIN {X -0.283,Y -609.349,Z 910.304,A 0.000,B 0.000,C 90.000,E1 270.745} C_DIS
LIN {X -0.106,Y -602.627,Z 910.302,A 0.000,B 0.000,C 90.000,E1 270.401} C_DIS
LIN {X -0.158,Y -597.555,Z 910.301,A 0.000,B 0.000,C 90.000,E1 270.172} C_DIS
LIN {X -0.149,Y -590.201,Z 910.299,A 0.000,B 0.000,C 90.000,E1 269.885} C_DIS
LIN {X 0.277,Y -584.770,Z 910.298,A 0.000,B 0.000,C 90.000,E1 269.656} C_DIS
LIN {X -0.204,Y -577.251,Z 910.297,A 0.000,B 0.000,C 90.000,E1 269.484} C_DIS
LIN {X 0.188,Y -571.273,Z 910.296,A 0.000,B 0.000,C 90.000,E1 269.312} C_DIS
LIN {X 0.252,Y -564.307,Z 910.296,A 0.000,B 0.000,C 90.000,E1 269.198} C_DIS
LIN {X -0.234,Y -552.333,Z 910.295,A 0.000,B 0.000,C 90.000,E1 269.141} C_DIS
LIN {X 0.065,Y -549.436,Z 910.295,A 0.000,B 0.000,C 90.000,E1 269.026} C_DIS
LIN {X 0.034,Y -549.322,Z 910.295,A 0.000,B 0.000,C 90.000,E1 269.026} C_DIS
LIN {X -0.001,Y -545.300,Z 910.293,A 0.000,B 0.000,C 90.000,E1 268.682} C_DIS
LIN {X -0.038,Y -545.267,Z 910.293,A 0.000,B 0.000,C 90.000,E1 268.682} C_DIS
LIN {X 0.189,Y -544.124,Z 910.291,A 0.000,B 0.000,C 90.000,E1 268.339} C_DIS
LIN {X 0.048,Y -542.893,Z 910.285,A 0.000,B 0.000,C 90.000,E1 267.364} C_DIS
LIN {X -0.122,Y -540.270,Z 910.268,A 0.000,B 0.000,C 90.000,E1 264.261} C_DIS
LIN {X 0.075,Y -539.276,Z 910.260,A 0.000,B 0.000,C 90.000,E1 262.818} C_DIS
LIN {X -0.285,Y -538.043,Z 910.252,A 0.000,B 0.000,C 90.000,E1 261.432} C_DIS
LIN {X -0.059,Y -536.690,Z 910.244,A 0.000,B 0.000,C 90.000,E1 259.982} C_DIS
LIN {X 0.236,Y -535.157,Z 910.236,A 0.000,B 0.000,C 90.000,E1 258.522} C_DIS
LIN {X 0.025,Y -533.118,Z 910.227,A 0.000,B 0.000,C 90.000,E1 256.825} C_DIS
LIN {X 0.022,Y -531.007,Z 910.217,A 0.000,B 0.000,C 90.000,E1 255.102} C_DIS
LIN {X 0.001,Y -528.503,Z 910.206,A 0.000,B 0.000,C 90.000,E1 253.087} C_DIS
LIN {X -0.132,Y -527.082,Z 910.200,A 0.000,B 0.000,C 90.000,E1 251.945} C_DIS
LIN {X 0.045,Y -524.792,Z 910.190,A 0.000,B 0.000,C 90.000,E1 250.188} C_DIS
LIN {X 0.190,Y -522.917,Z 910.182,A 0.000,B 0.000,C 90.000,E1 248.720} C_DIS
LIN {X 0.011,Y -520.892,Z 910.174,A 0.000,B 0.000,C 90.000,E1 247.283} C_DIS
LIN {X 0.135,Y -519.297,Z 910.167,A 0.000,B 0.000,C 90.000,E1 246.102} C_DIS
LIN {X 0.036,Y -515.800,Z 910.154,A 0.000,B 0.000,C 90.000,E1 243.768} C_DIS
LIN {X -0.169,Y -512.889,Z 910.145,A 0.000,B 0.000,C 90.000,E1 242.025} C_DIS
LIN {X -0.073,Y -511.346,Z 910.140,A 0.000,B 0.000,C 90.000,E1 241.129} C_DIS
LIN {X -0.252,Y -507.618,Z 910.128,A 0.000,B 0.000,C 90.000,E1 239.076} C_DIS
LIN {X 0.290,Y -506.035,Z 910.123,A 0.000,B 0.000,C 90.000,E1 238.122} C_DIS
LIN {X 0.006,Y -503.687,Z 910.117,A 0.000,B 0.000,C 90.000,E1 236.962} C_DIS
LIN {X 0.103,Y -501.209,Z 910.110,A 0.000,B 0.000,C 90.000,E1 235.754} C_DIS
LIN {X -0.137,Y -499.861,Z 910.107,A 0.000,B 0.000,C 90.000,E1 235.182} C_DIS
LIN {X -0.232,Y -497.095,Z 910.100,A 0.000,B 0.000,C 90.000,E1 233.989} C_DIS
LIN {X 0.063,Y -495.088,Z 910.095,A 0.000,B 0.000,C 90.000,E1 233.050} C_DIS
LIN {X 0.044,Y -491.735,Z 910.086,A 0.000,B 0.000,C 90.000,E1 231.537} C_DIS
LIN {X 0.263,Y -488.277,Z 910.078,A 0.000,B 0.000,C 90.000,E1 229.989} C_DIS
LIN {X 0.040,Y -484.998,Z 910.069,A 0.000,B 0.000,C 90.000,E1 228.485} C_DIS
LIN {X -0.226,Y -479.473,Z 910.056,A 0.000,B 0.000,C 90.000,E1 226.053} C_DIS
LIN {X 0.025,Y -475.978,Z 910.047,A 0.000,B 0.000,C 90.000,E1 224.474} C_DIS
LIN {X -0.115,Y -472.396,Z 910.039,A 0.000,B 0.000,C 90.000,E1 222.933} C_DIS
LIN {X 0.192,Y -467.490,Z 910.026,A 0.000,B 0.000,C 90.000,E1 220.701} C_DIS
LIN {X 0.249,Y -464.160,Z 910.018,A 0.000,B 0.000,C 90.000,E1 219.116} C_DIS
LIN {X 0.056,Y -460.112,Z 910.007,A 0.000,B 0.000,C 90.000,E1 217.237} C_DIS
LIN {X 0.035,Y -456.737,Z 909.998,A 0.000,B 0.000,C 90.000,E1 215.644} C_DIS
LIN {X 0.047,Y -453.349,Z 909.989,A 0.000,B 0.000,C 90.000,E1 214.040} C_DIS
LIN {X -0.018,Y -447.567,Z 909.975,A 0.000,B 0.000,C 90.000,E1 211.465} C_DIS
LIN {X 0.199,Y -445.434,Z 909.969,A 0.000,B 0.000,C 90.000,E1 210.463} C_DIS
LIN {X -0.059,Y -441.147,Z 909.959,A 0.000,B 0.000,C 90.000,E1 208.537} C_DIS
LIN {X 0.116,Y -437.567,Z 909.949,A 0.000,B 0.000,C 90.000,E1 206.873} C_DIS
LIN {X 0.043,Y -433.225,Z 909.938,A 0.000,B 0.000,C 90.000,E1 204.899} C_DIS
LIN {X -0.122,Y -429.573,Z 909.929,A 0.000,B 0.000,C 90.000,E1 203.259} C_DIS
LIN {X -0.136,Y -426.013,Z 909.920,A 0.000,B 0.000,C 90.000,E1 201.589} C_DIS
LIN {X -0.006,Y -421.033,Z 909.907,A 0.000,B 0.000,C 90.000,E1 199.214} C_DIS
LIN {X 0.092,Y -417.030,Z 909.896,A 0.000,B 0.000,C 90.000,E1 197.166} C_DIS
LIN {X -0.030,Y -412.916,Z 909.884,A 0.000,B 0.000,C 90.000,E1 195.134} C_DIS
LIN {X 0.035,Y -408.759,Z 909.873,A 0.000,B 0.000,C 90.000,E1 193.063} C_DIS
LIN {X -0.190,Y -405.355,Z 909.863,A 0.000,B 0.000,C 90.000,E1 191.366} C_DIS
LIN {X -0.087,Y -401.905,Z 909.853,A 0.000,B 0.000,C 90.000,E1 189.613} C_DIS
LIN {X -0.132,Y -398.413,Z 909.844,A 0.000,B 0.000,C 90.000,E1 187.871} C_DIS
LIN {X -0.157,Y -392.386,Z 909.826,A 0.000,B 0.000,C 90.000,E1 184.702} C_DIS
LIN {X 0.073,Y -388.147,Z 909.812,A 0.000,B 0.000,C 90.000,E1 182.178} C_DIS
LIN {X -0.108,Y -384.614,Z 909.800,A 0.000,B 0.000,C 90.000,E1 180.057} C_DIS
LIN {X -0.107,Y -380.799,Z 909.786,A 0.000,B 0.000,C 90.000,E1 177.535} C_DIS
LIN {X 0.171,Y -378.775,Z 909.778,A 0.000,B 0.000,C 90.000,E1 176.045} C_DIS
LIN {X -0.176,Y -377.624,Z 909.772,A 0.000,B 0.000,C 90.000,E1 175.008} C_DIS
LIN {X -0.048,Y -377.269,Z 909.768,A 0.000,B 0.000,C 90.000,E1 174.261} C_DIS
LIN {X 0.042,Y -377.175,Z 909.763,A 0.000,B 0.000,C 90.000,E1 173.337} C_DIS
LIN {X -0.034,Y -377.855,Z 909.759,A 0.000,B 0.000,C 90.000,E1 172.591} C_DIS
LIN {X -0.008,Y -379.397,Z 909.755,A 0.000,B 0.000,C 90.000,E1 171.837} C_DIS
LIN {X -0.124,Y -381.316,Z 909.752,A 0.000,B 0.000,C 90.000,E1 171.310} C_DIS
LIN {X 0.179,Y -381.805,Z 909.751,A 0.000,B 0.000,C 90.000,E1 171.084} C_DIS
LIN {X 0.083,Y -385.104,Z 909.748,A 0.000,B 0.000,C 90.000,E1 170.557} C_DIS
LIN {X 0.032,Y -387.151,Z 909.746,A 0.000,B 0.000,C 90.000,E1 170.274} C_DIS
LIN {X -0.041,Y -390.471,Z 909.744,A 0.000,B 0.000,C 90.000,E1 169.926} C_DIS
LIN {X 0.163,Y -394.797,Z 909.742,A 0.000,B 0.000,C 90.000,E1 169.511} C_DIS
LIN {X 0.025,Y -403.623,Z 909.739,A 0.000,B 0.000,C 90.000,E1 168.926} C_DIS
LIN {X -0.013,Y -417.027,Z 909.734,A 0.000,B 0.000,C 90.000,E1 168.049} C_DIS
LIN {X 0.118,Y -423.325,Z 909.731,A 0.000,B 0.000,C 90.000,E1 167.589} C_DIS
LIN {X 0.145,Y -429.742,Z 909.729,A 0.000,B 0.000,C 90.000,E1 167.117} C_DIS
LIN {X -0.093,Y -439.194,Z 909.724,A 0.000,B 0.000,C 90.000,E1 166.408} C_DIS
LIN {X 0.194,Y -443.639,Z 909.722,A 0.000,B 0.000,C 90.000,E1 165.992} C_DIS
LIN {X 0.029,Y -452.607,Z 909.718,A 0.000,B 0.000,C 90.000,E1 165.227} C_DIS
LIN {X 0.133,Y -461.184,Z 909.713,A 0.000,B 0.000,C 90.000,E1 164.393} C_DIS
LIN {X -0.174,Y -472.263,Z 909.707,A 0.000,B 0.000,C 90.000,E1 163.268} C_DIS
LIN {X -0.089,Y -477.679,Z 909.704,A 0.000,B 0.000,C 90.000,E1 162.670} C_DIS
LIN {X 0.168,Y -483.985,Z 909.699,A 0.000,B 0.000,C 90.000,E1 161.873} C_DIS
LIN {X 0.291,Y -492.612,Z 909.693,A 0.000,B 0.000,C 90.000,E1 160.786} C_DIS
LIN {X 0.206,Y -497.235,Z 909.690,A 0.000,B 0.000,C 90.000,E1 160.188} C_DIS
LIN {X 0.104,Y -506.988,Z 909.683,A 0.000,B 0.000,C 90.000,E1 158.847} C_DIS
LIN {X 0.010,Y -510.108,Z 909.680,A 0.000,B 0.000,C 90.000,E1 158.411} C_DIS
LIN {X 0.067,Y -518.098,Z 909.674,A 0.000,B 0.000,C 90.000,E1 157.230} C_DIS
LIN {X -0.143,Y -524.939,Z 909.668,A 0.000,B 0.000,C 90.000,E1 156.230} C_DIS
LIN {X -0.231,Y -534.278,Z 909.660,A 0.000,B 0.000,C 90.000,E1 154.793} C_DIS
LIN {X -0.012,Y -540.422,Z 909.654,A 0.000,B 0.000,C 90.000,E1 153.768} C_DIS
LIN {X 0.041,Y -548.035,Z 909.647,A 0.000,B 0.000,C 90.000,E1 152.487} C_DIS
LIN {X -0.278,Y -554.962,Z 909.640,A 0.000,B 0.000,C 90.000,E1 151.257} C_DIS
LIN {X -0.116,Y -560.683,Z 909.634,A 0.000,B 0.000,C 90.000,E1 150.127} C_DIS
LIN {X -0.060,Y -567.577,Z 909.626,A 0.000,B 0.000,C 90.000,E1 148.742} C_DIS
LIN {X -0.113,Y -572.180,Z 909.621,A 0.000,B 0.000,C 90.000,E1 147.788} C_DIS
LIN {X -0.192,Y -577.306,Z 909.615,A 0.000,B 0.000,C 90.000,E1 146.707} C_DIS
LIN {X -0.041,Y -583.295,Z 909.607,A 0.000,B 0.000,C 90.000,E1 145.341} C_DIS
LIN {X -0.134,Y -587.894,Z 909.602,A 0.000,B 0.000,C 90.000,E1 144.276} C_DIS
LIN {X -0.015,Y -591.287,Z 909.597,A 0.000,B 0.000,C 90.000,E1 143.463} C_DIS
LIN {X 0.013,Y -595.564,Z 909.591,A 0.000,B 0.000,C 90.000,E1 142.396} C_DIS
LIN {X -0.118,Y -603.006,Z 909.581,A 0.000,B 0.000,C 90.000,E1 140.561} C_DIS
LIN {X 0.046,Y -609.518,Z 909.572,A 0.000,B 0.000,C 90.000,E1 138.976} C_DIS
LIN {X 0.014,Y -618.199,Z 909.561,A 0.000,B 0.000,C 90.000,E1 136.905} C_DIS
LIN {X 0.011,Y -624.781,Z 909.552,A 0.000,B 0.000,C 90.000,E1 135.364} C_DIS
LIN {X 0.183,Y -626.996,Z 909.549,A 0.000,B 0.000,C 90.000,E1 134.838} C_DIS
LIN {X 0.023,Y -632.256,Z 909.542,A 0.000,B 0.000,C 90.000,E1 133.581} C_DIS
LIN {X -0.047,Y -637.481,Z 909.535,A 0.000,B 0.000,C 90.000,E1 132.324} C_DIS
LIN {X -0.038,Y -642.576,Z 909.528,A 0.000,B 0.000,C 90.000,E1 131.067} C_DIS
